(* CODESYS project CÓDIGO FINAL - Separação de caixas coloridas.project

Project tree, tasks and I/O mapping:
  Device : CODESYS Control Win V3, 3S - Smart Software Solutions GmbH, order no. 305021, version 3.5.11.30
    application Application
      libraries: Standard, * (System)
      task MainTask (cyclic, interval t#20ms, priority 1) calls VACUO_01, VACUO_02, PALETIZADOR_01, PALETIZADOR_02, ESTOCAGEM_01, ESTOCAGEM_02
      program VACUO_01 [LD]
      Symbols
      program VACUO_02 [LD]
      global variables MY_GLOBAL
      program PALETIZADOR_01 [LD]
      program PALETIZADOR_02 [LD]
      program ESTOCAGEM_01 [LD]
      program ESTOCAGEM_02 [LD]
*)

// Device/Application/MY_GLOBAL
{attribute 'qualified_only'}
VAR_GLOBAL
// 	VARIAVEL GLOBAL
 	CONTROLE:BOOL;
END_VAR

// Device/Application/VACUO_01
PROGRAM VACUO_01
VAR
// PAINEL DE CONTROLE 
	//ENTRADAS
	_START:BOOL;
	_STOP:BOOL;
	_RESET:BOOL;
	_EMERGENCIA_STOP:BOOL;
	
	//SAIDAS
	START_LIGHT:BOOL;
	STOP_LIGHT:BOOL;
	RESET_LIGHT:BOOL;
	RED: BOOL;
	GREEN: BOOL;
	YELLOW: BOOL;
	CONTAGEM_VERDES:UINT;
	CONTAGEM_DEFEITOS: UINT;
	
// ESTEIRA PRINCIPAL
	//ENTRADAS
	_SENSOR_CAIXA:REAL;
	
	//SAIDAS
	ESTEIRA_PRINCIPAL:BOOL;
	ESTEIRA_PRINCIPAL_1:BOOL;

// ESTEIRA SECUDARIA N 01(VERDE)
	//ENTRADAS
	_SENSOR_SAIDA01:BOOL;
	
	//SAIDAS
	ESTEIRA_SECUDARIA01:BOOL;
	ESTEIRA_CURVA_SECUNDARIA1:BOOL;
	ESTEIRA_CURVA_SECUNDARIA1_1:BOOL;
	ESTEIRA_SAIDA_PALETE1: BOOL;
	
// VACUO N 01
	//ENTRADAS
	_SENSOR_ENTRADA01:BOOL;
	_DETECTED_VACUO01:BOOL;
	
	//SAIDAS
	X1:BOOL;
	Y1:BOOL;
	VACUO_1:BOOL;
	
// AUXILIARES
	CAIXA_VERDE: BOOL;
	A1: BOOL;
	A2: BOOL;
	A3: BOOL;
	A4: BOOL;
	A5: BOOL;
	A6: BOOL;
	A7: BOOL;
	A8: BOOL;
	A9: BOOL;
	A10: BOOL;
	A11: BOOL;

//TEMPORIZADORES
	TON_1A: TON;
	TEMPO_1A: TIME;
	TON_2A: TON;
	TEMPO_2A: TIME;
	TON_3A: TON;
	TEMPO_3A: TIME;
	TON_4A: TON;
	TEMPO_4A: TIME;
	TON_5A: TON;
	TEMPO_5A: TIME;
	TON_6A: TON;
	TEMPO_6A: TIME;
	TON_7A: TON;
	TEMPO_7A: TIME;
	TON_8A: TON;
	TEMPO_8A: TIME;
	TON_9A: TON;
	TEMPO_9A: TIME;
	TON_10A: TON;
	TEMPO_10A: TIME;
	TON_11A: TON;
	TEMPO_11A: TIME;

//CONTADORES
	CTU_1A: CTU;
	CONT_1A: WORD;
	CTU_2A: CTU;
	CONT_2A: WORD;
END_VAR
VAR // added by the converter: edge detectors and wires of the graphical bodies
    _w1, _w2, _w3, _w4, _w5, _w6, _w7, _w8, _w9 : BOOL;
END_VAR

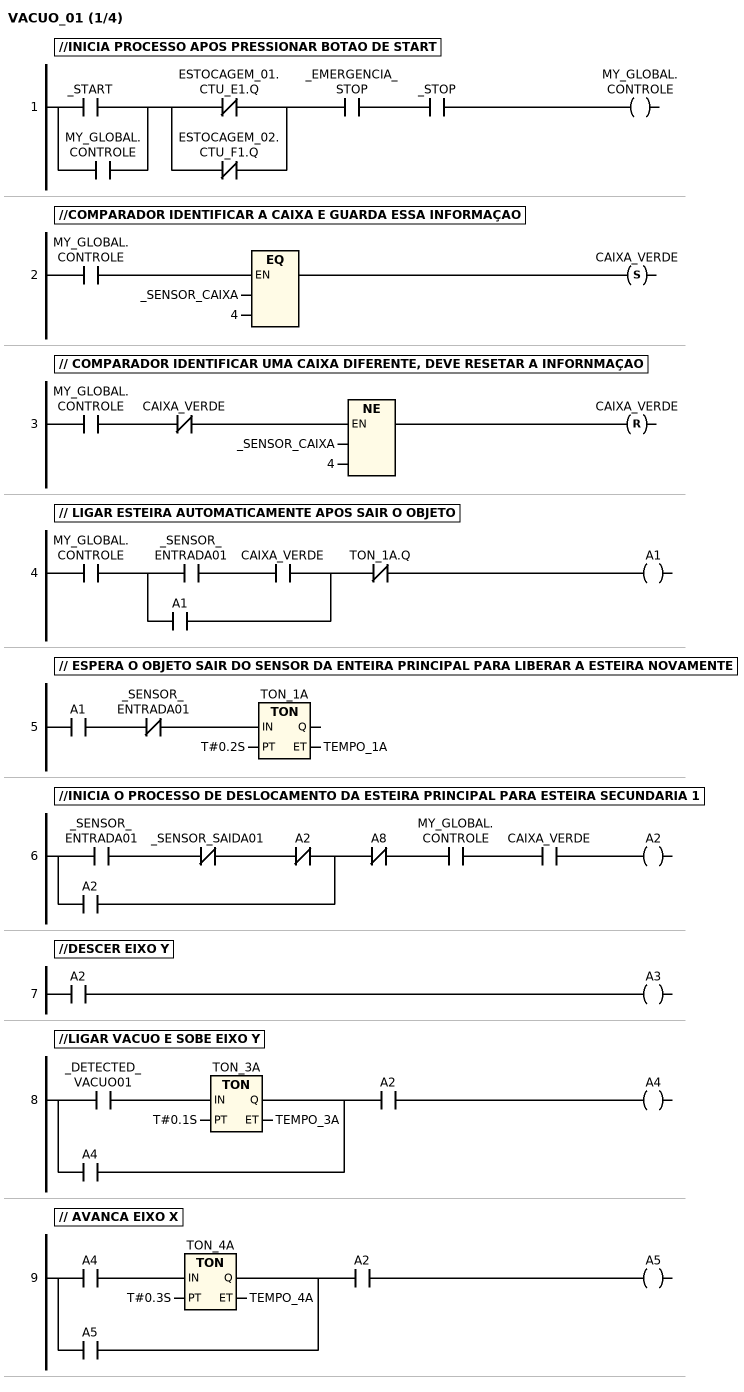
// NETWORK 1
// label: //INICIA PROCESSO APOS PRESSIONAR BOTAO DE START
MY_GLOBAL.CONTROLE := (_START OR MY_GLOBAL.CONTROLE) AND (NOT ESTOCAGEM_01.CTU_E1.Q OR NOT ESTOCAGEM_02.CTU_F1.Q) AND _EMERGENCIA_STOP AND _STOP;

// NETWORK 2
// label: //COMPARADOR IDENTIFICAR A CAIXA E GUARDA ESSA INFORMAÇAO
CAIXA_VERDE S= MY_GLOBAL.CONTROLE AND _SENSOR_CAIXA = 4;

// NETWORK 3
// label: // COMPARADOR IDENTIFICAR UMA CAIXA DIFERENTE, DEVE RESETAR A INFORNMAÇAO
CAIXA_VERDE R= MY_GLOBAL.CONTROLE AND NOT CAIXA_VERDE AND _SENSOR_CAIXA <> 4;

// NETWORK 4
// label: // LIGAR ESTEIRA AUTOMATICAMENTE APOS SAIR O OBJETO
A1 := MY_GLOBAL.CONTROLE AND (_SENSOR_ENTRADA01 AND CAIXA_VERDE OR A1) AND NOT TON_1A.Q;

// NETWORK 5
// label: // ESPERA O OBJETO SAIR DO SENSOR DA ENTEIRA PRINCIPAL PARA LIBERAR A ESTEIRA NOVAMENTE
TON_1A(IN := A1 AND NOT _SENSOR_ENTRADA01, PT := T#0.2S, ET => TEMPO_1A); // TON

// NETWORK 6
// label: //INICIA O PROCESSO DE DESLOCAMENTO DA ESTEIRA PRINCIPAL PARA ESTEIRA SECUNDARIA 1
A2 := (_SENSOR_ENTRADA01 AND NOT _SENSOR_SAIDA01 AND NOT A2 OR A2) AND NOT A8 AND MY_GLOBAL.CONTROLE AND CAIXA_VERDE;

// NETWORK 7
// label: //DESCER EIXO Y
A3 := A2;

// NETWORK 8
// label: //LIGAR VACUO E SOBE EIXO Y
TON_3A(IN := _DETECTED_VACUO01, PT := T#0.1S, ET => TEMPO_3A); // TON
A4 := (TON_3A.Q OR A4) AND A2;

// NETWORK 9
// label: // AVANCA EIXO X
TON_4A(IN := A4, PT := T#0.3S, ET => TEMPO_4A); // TON
A5 := (TON_4A.Q OR A5) AND A2;

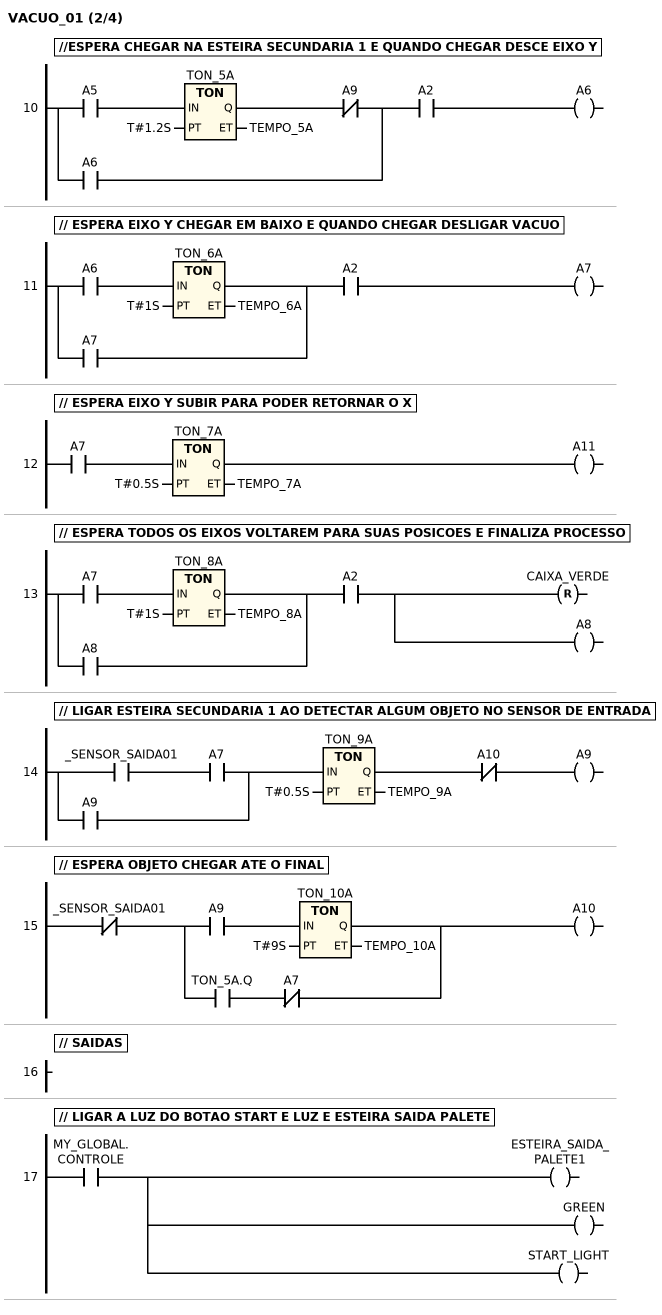
// NETWORK 10
// label: //ESPERA CHEGAR NA ESTEIRA SECUNDARIA 1 E QUANDO CHEGAR DESCE EIXO Y
TON_5A(IN := A5, PT := T#1.2S, ET => TEMPO_5A); // TON
A6 := (TON_5A.Q AND NOT A9 OR A6) AND A2;

// NETWORK 11
// label: // ESPERA EIXO Y CHEGAR EM BAIXO E QUANDO CHEGAR DESLIGAR VACUO
TON_6A(IN := A6, PT := T#1S, ET => TEMPO_6A); // TON
A7 := (TON_6A.Q OR A7) AND A2;

// NETWORK 12
// label: // ESPERA EIXO Y SUBIR PARA PODER RETORNAR O X
TON_7A(IN := A7, PT := T#0.5S, ET => TEMPO_7A); // TON
A11 := TON_7A.Q;

// NETWORK 13
// label: // ESPERA TODOS OS EIXOS VOLTAREM PARA SUAS POSICOES E FINALIZA PROCESSO
TON_8A(IN := A7, PT := T#1S, ET => TEMPO_8A); // TON
_w1 := (TON_8A.Q OR A8) AND A2;
CAIXA_VERDE R= _w1;
A8 := _w1;

// NETWORK 14
// label: // LIGAR ESTEIRA SECUNDARIA 1 AO DETECTAR ALGUM OBJETO NO SENSOR DE ENTRADA
TON_9A(IN := _SENSOR_SAIDA01 AND A7 OR A9, PT := T#0.5S, ET => TEMPO_9A); // TON
A9 := TON_9A.Q AND NOT A10;

// NETWORK 15
// label: // ESPERA OBJETO CHEGAR ATE O FINAL
_w2 := NOT _SENSOR_SAIDA01;
_w3 := (_w2 AND TON_5A.Q) AND NOT A7;
IF NOT _w3 THEN
    TON_10A(IN := _w2 AND A9, PT := T#9S, ET => TEMPO_10A); // TON
    _w3 := TON_10A.Q;
END_IF
A10 := _w3;

// NETWORK 16
// label: // SAIDAS

// NETWORK 17
// label: // LIGAR A LUZ DO BOTAO START E LUZ E ESTEIRA SAIDA PALETE
ESTEIRA_SAIDA_PALETE1 := MY_GLOBAL.CONTROLE;
GREEN := MY_GLOBAL.CONTROLE;
START_LIGHT := MY_GLOBAL.CONTROLE;

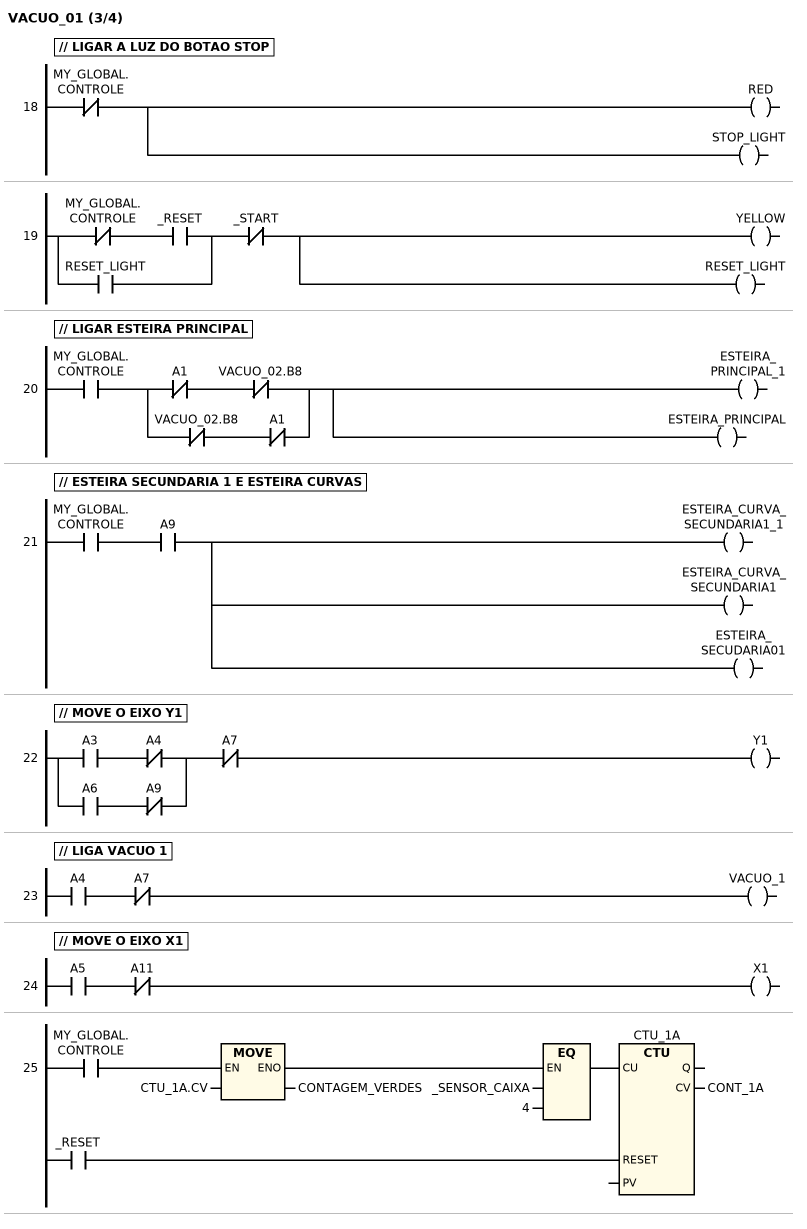
// NETWORK 18
// label: // LIGAR A LUZ DO BOTAO STOP
_w4 := NOT MY_GLOBAL.CONTROLE;
RED := _w4;
STOP_LIGHT := _w4;

// NETWORK 19
_w5 := (NOT MY_GLOBAL.CONTROLE AND _RESET OR RESET_LIGHT) AND NOT _START;
YELLOW := _w5;
RESET_LIGHT := _w5;

// NETWORK 20
// label: // LIGAR ESTEIRA PRINCIPAL
_w6 := MY_GLOBAL.CONTROLE AND (NOT A1 AND NOT VACUO_02.B8 OR NOT VACUO_02.B8 AND NOT A1);
ESTEIRA_PRINCIPAL_1 := _w6;
ESTEIRA_PRINCIPAL := _w6;

// NETWORK 21
// label: // ESTEIRA SECUNDARIA 1 E ESTEIRA CURVAS
_w7 := MY_GLOBAL.CONTROLE AND A9;
ESTEIRA_CURVA_SECUNDARIA1_1 := _w7;
ESTEIRA_CURVA_SECUNDARIA1 := _w7;
ESTEIRA_SECUDARIA01 := _w7;

// NETWORK 22
// label: // MOVE O EIXO Y1
Y1 := (A3 AND NOT A4 OR A6 AND NOT A9) AND NOT A7;

// NETWORK 23
// label: // LIGA VACUO 1
VACUO_1 := A4 AND NOT A7;

// NETWORK 24
// label: // MOVE O EIXO X1
X1 := A5 AND NOT A11;

// NETWORK 25
_w8 := MY_GLOBAL.CONTROLE;
IF _w8 THEN CONTAGEM_VERDES := CTU_1A.CV; END_IF
CTU_1A(CU := _w8 AND _SENSOR_CAIXA = 4, RESET := _RESET, CV => CONT_1A); // CTU

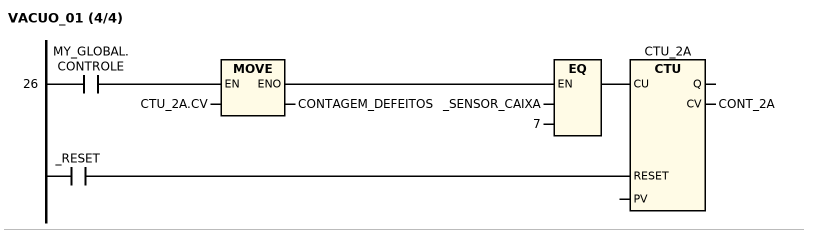
// NETWORK 26
_w9 := MY_GLOBAL.CONTROLE;
IF _w9 THEN CONTAGEM_DEFEITOS := CTU_2A.CV; END_IF
CTU_2A(CU := _w9 AND _SENSOR_CAIXA = 7, RESET := _RESET, CV => CONT_2A); // CTU

END_PROGRAM

// Device/Application/ESTOCAGEM_01
PROGRAM ESTOCAGEM_01
VAR
//ENTRADA
	_SENSOR_ESTOCAGEM1: BOOL;

//SAIDA
	CRANE_ENTRADA1:BOOL;
	CRANE_SAIDA1:BOOL;
	CRANE_SUBIR1:BOOL;
	ESTEIRA_ESTOCAGEM1:BOOL;
	ESTEIRA_MEIO_ESTOCAGEM1:BOOL;
	ESTEIRA_CURVA_ESTOCAGEM1:BOOL;
	POSICAO: UINT;
//AUXILIARES	
	E1: BOOL;
	E2: BOOL;
	E3: BOOL;
	E4: BOOL;
	E5: BOOL;	

//TEMPORIZAODES 
	TON_E1: TON;
	TEMPO_E1: TIME;
	TON_E2: TON;
	TEMPO_E2: TIME;
	TON_E3: TON;
	TEMPO_E3: TIME;
	TON_E4: TON;
	TEMPO_E4: TIME;
	TON_E5: TON;
	TEMPO_E5: TIME;
	TON_E6: TON;
	TEMPO_E6: TIME;

//CONTADORES
	CTU_E1: CTU;
	CONT_E1: WORD;

// TEMPORIZADORES DE CADA PRATILEIRA
	TON_1:TON;
	TEMPO_1:TIME;
	TON_2:TON;
	TEMPO_2:TIME;
	TON_3:TON;
	TEMPO_3: TIME;
	TON_4:TON;
	TEMPO_4:TIME;
	TON_5:TON;
	TEMPO_5:TIME;
	TON_6:TON;
	TEMPO_6:TIME;
	TON_7:TON;
	TEMPO_7:TIME;
	TON_8:TON;
	TEMPO_8:TIME;
	TON_9:TON;
	TEMPO_9:TIME;
	TON_10: TON;
	TEMPO_10: TIME;
	TON_11: TON;
	TEMPO_11: TIME;
	TON_12: TON;
	TEMPO_12: TIME;
	TON_13:TON;
	TEMPO_13: TIME;
	TON_14: TON;
	TEMPO_14: TIME;
	TON_15: TON;
	TEMPO_15: TIME;
	TON_16: TON;
	TEMPO_16: TIME;
	TON_17: TON;
	TEMPO_17: TIME;
	TON_18: TON;
	TEMPO_18: TIME;
	TON_19: TON;
	TEMPO_19: TIME;
	TON_20: TON;
	TEMPO_20: TIME;
	TON_21: TON;
	TEMPO_21: TIME;
	TON_22: TON;
	TEMPO_22: TIME;
	TON_23: TON;
	TEMPO_23: TIME;
	TON_24: TON;
	TEMPO_24: TIME;
	TON_25: TON;
	TEMPO_25: TIME;
	TON_26: TON;
	TEMPO_26: TIME;
	TON_27: TON;
	TEMPO_27: TIME;
	TON_28: TON;
	TEMPO_28: TIME;
	TON_29: TON;
	TEMPO_29: TIME;
	TON_30: TON;
	TEMPO_30: TIME;
	TON_31: TON;
	TEMPO_31: TIME;
	TON_32: TON;
	TEMPO_32: TIME;
	TON_33: TON;
	TEMPO_33: TIME;
	TON_34: TON;
	TEMPO_34: TIME;
	TON_35: TON;
	TEMPO_35: TIME;
	TON_36: TON;
	TEMPO_36: TIME;
	TON_37: TON;
	TEMPO_37: TIME;
	TON_38: TON;
	TEMPO_38: TIME;
	TON_39: TON;
	TEMPO_39: TIME;
	TON_40: TON;
	TEMPO_40: TIME;
	TON_41: TON;
	TEMPO_41: TIME;
	TON_42: TON;
	TEMPO_42: TIME;
	TON_43: TON;
	TEMPO_43: TIME;
	TON_44: TON;
	TEMPO_44: TIME;
	TON_45: TON;
	TEMPO_45: TIME;
	TON_46: TON;
	TEMPO_46: TIME;
	TON_47: TON;
	TEMPO_47: TIME;
	TON_48: TON;
	TEMPO_48: TIME;
	TON_49: TON;
	TEMPO_49: TIME;
	TON_50: TON;
	TEMPO_50: TIME;
	TON_51: TON;
	TEMPO_51: TIME;
	TON_52: TON;
	TEMPO_52: TIME;
	TON_53: TON;
	TEMPO_53: TIME;
	TON_54: TON;
	TEMPO_54: TIME;

// AUXILIARES DE CADA PRATILEIRA
	T1:BOOL;
	T2:BOOL;
	T3:BOOL;
	T4:BOOL;
	T5:BOOL;
	T6:BOOL;
	T7:BOOL;
	T8:BOOL;
	T9:BOOL;
	T10:BOOL;
	T11:BOOL;
	T12:BOOL;
	T13:BOOL;
	T14:BOOL;
	T15:BOOL;
	T16:BOOL;
	T17:BOOL;
	T18:BOOL;	
	T19:BOOL;
	T20:BOOL;
	T21:BOOL;
	T22:BOOL;
	T23: BOOL;
	T24: BOOL;
	T25: BOOL;
	T26: BOOL;
	T27: BOOL;
	T28: BOOL;
	T29: BOOL;
	T30: BOOL;
	T31: BOOL;
	T32: BOOL;
	T33: BOOL;
	T34: BOOL;
	T35: BOOL;
	T36: BOOL;
	T37: BOOL;
	T38: BOOL;
	T39: BOOL;
	T40: BOOL;
	T41: BOOL;
	T42: BOOL;
	T43: BOOL;
	T44: BOOL;
	T45: BOOL;
	T46: BOOL;
	T47: BOOL;
	T48: BOOL;
	T49: BOOL;
	T50: BOOL;
	T51: BOOL;
	T52: BOOL;
	T53: BOOL;
	T54: BOOL;
	T55: BOOL;
END_VAR
VAR // added by the converter: edge detectors and wires of the graphical bodies
    _w1, _w2, _w3 : BOOL;
END_VAR

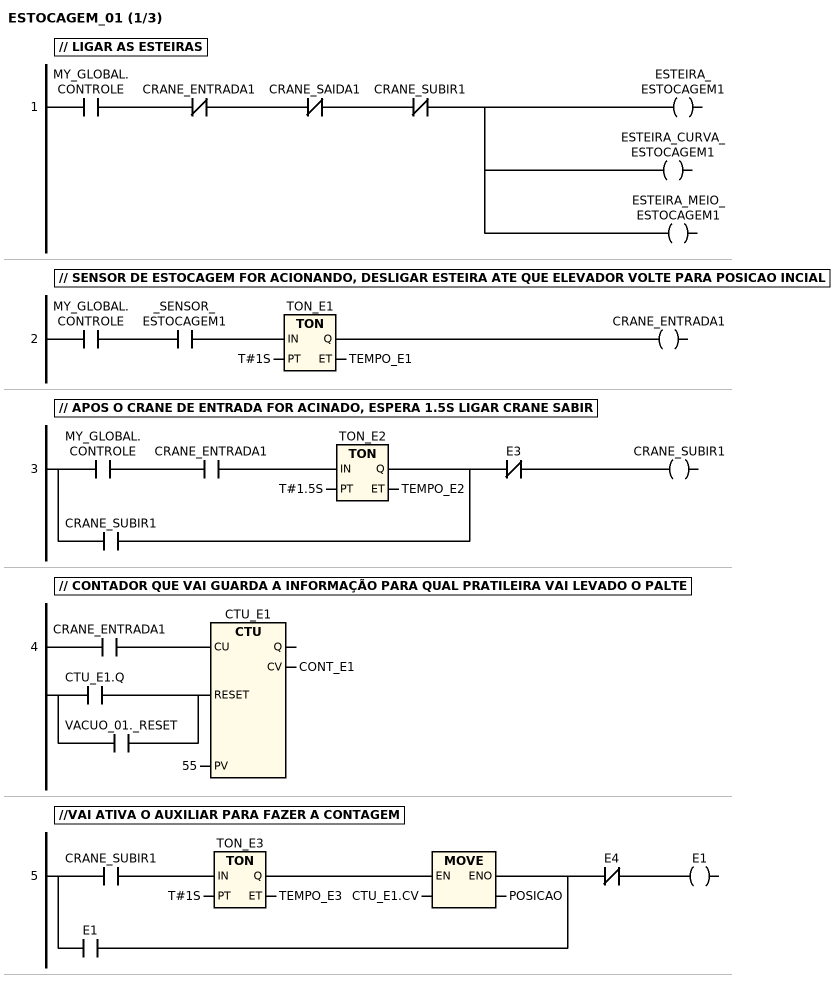
// NETWORK 1
// label: // LIGAR AS ESTEIRAS
_w1 := MY_GLOBAL.CONTROLE AND NOT CRANE_ENTRADA1 AND NOT CRANE_SAIDA1 AND NOT CRANE_SUBIR1;
ESTEIRA_ESTOCAGEM1 := _w1;
ESTEIRA_CURVA_ESTOCAGEM1 := _w1;
ESTEIRA_MEIO_ESTOCAGEM1 := _w1;

// NETWORK 2
// label: // SENSOR DE ESTOCAGEM FOR ACIONANDO, DESLIGAR ESTEIRA ATE QUE ELEVADOR VOLTE PARA POSICAO INCIAL
TON_E1(IN := MY_GLOBAL.CONTROLE AND _SENSOR_ESTOCAGEM1, PT := T#1S, ET => TEMPO_E1); // TON
CRANE_ENTRADA1 := TON_E1.Q;

// NETWORK 3
// label: // APOS O CRANE DE ENTRADA FOR ACINADO, ESPERA 1.5S LIGAR CRANE SABIR
TON_E2(IN := MY_GLOBAL.CONTROLE AND CRANE_ENTRADA1, PT := T#1.5S, ET => TEMPO_E2); // TON
CRANE_SUBIR1 := (TON_E2.Q OR CRANE_SUBIR1) AND NOT E3;

// NETWORK 4
// label: // CONTADOR QUE VAI GUARDA A INFORMAÇÃO PARA QUAL PRATILEIRA VAI LEVADO O PALTE
CTU_E1(CU := CRANE_ENTRADA1, RESET := CTU_E1.Q OR VACUO_01._RESET, PV := 55, CV => CONT_E1); // CTU

// NETWORK 5
// label: //VAI ATIVA O AUXILIAR PARA FAZER A CONTAGEM
TON_E3(IN := CRANE_SUBIR1, PT := T#1S, ET => TEMPO_E3); // TON
_w2 := TON_E3.Q;
IF _w2 THEN POSICAO := CTU_E1.CV; END_IF
E1 := (_w2 OR E1) AND NOT E4;

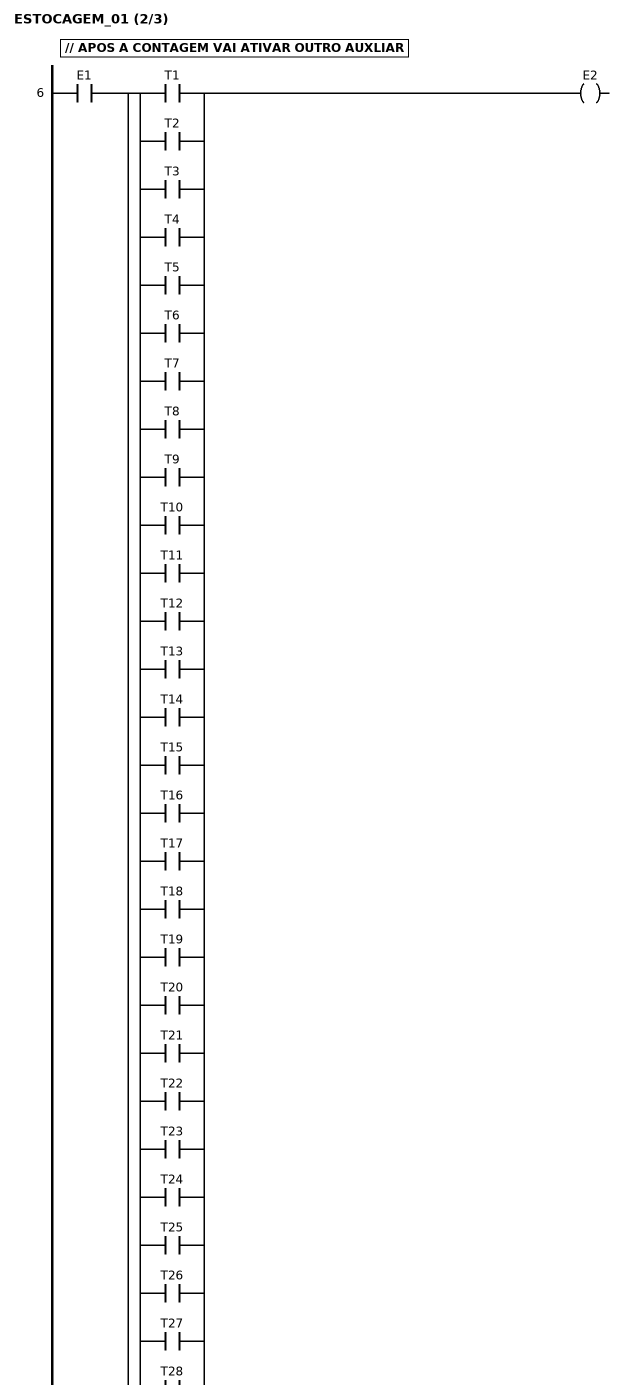
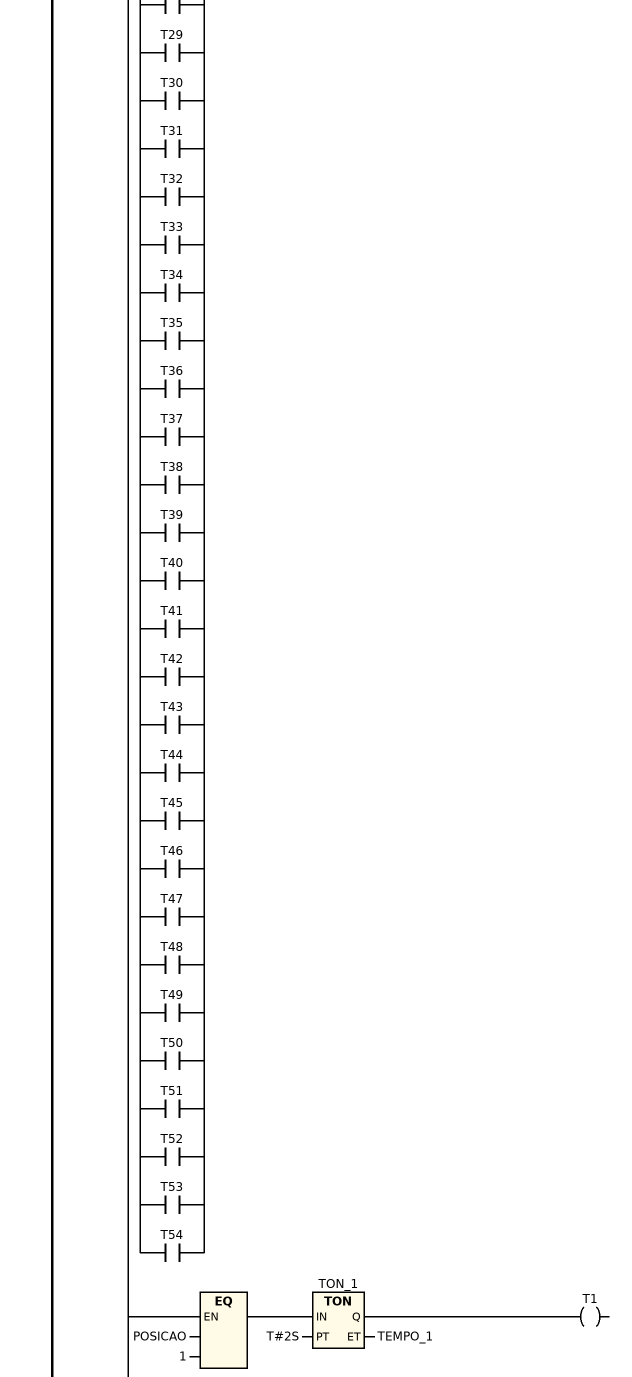
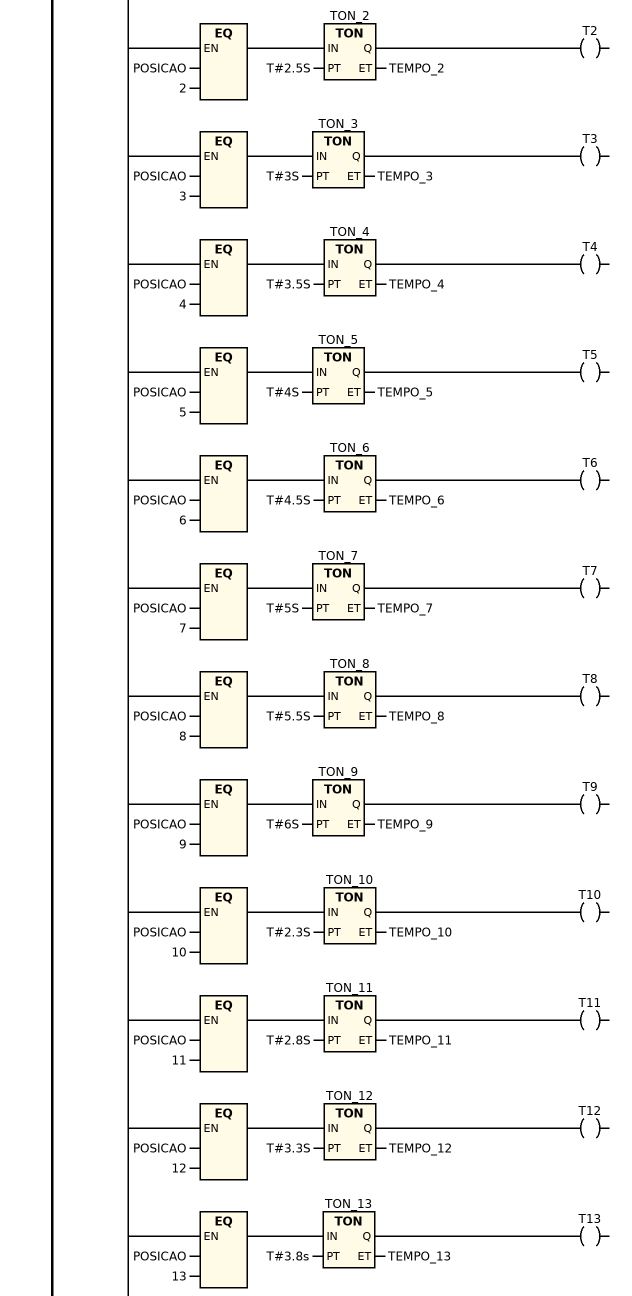
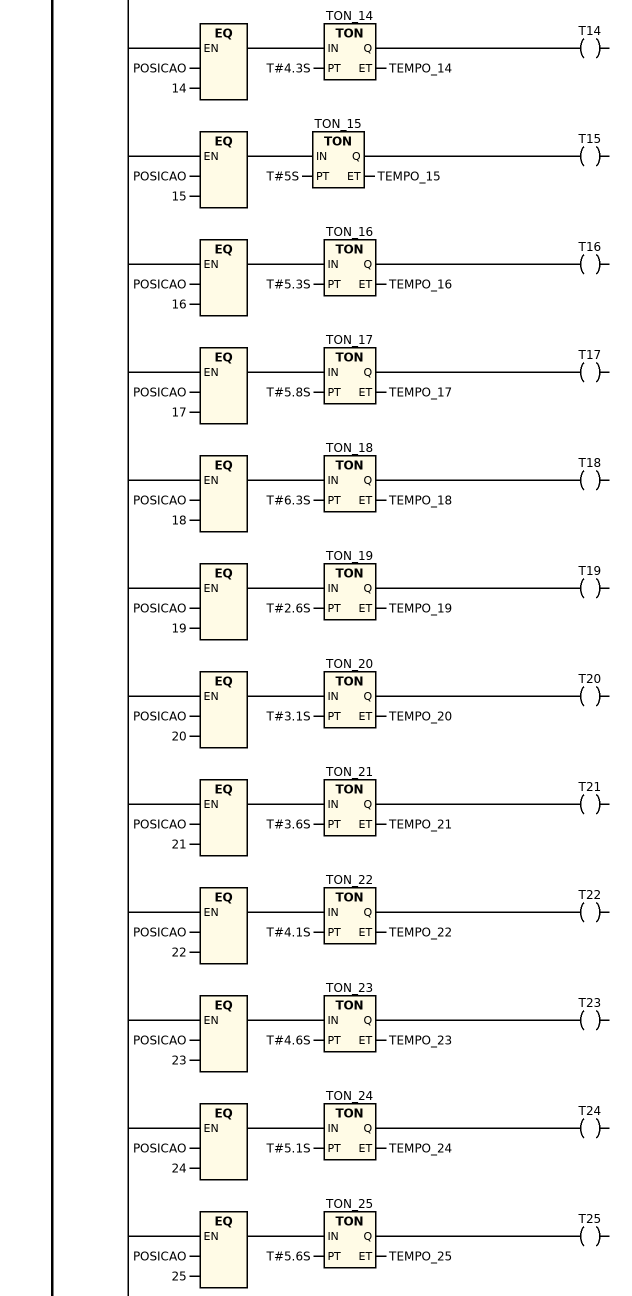
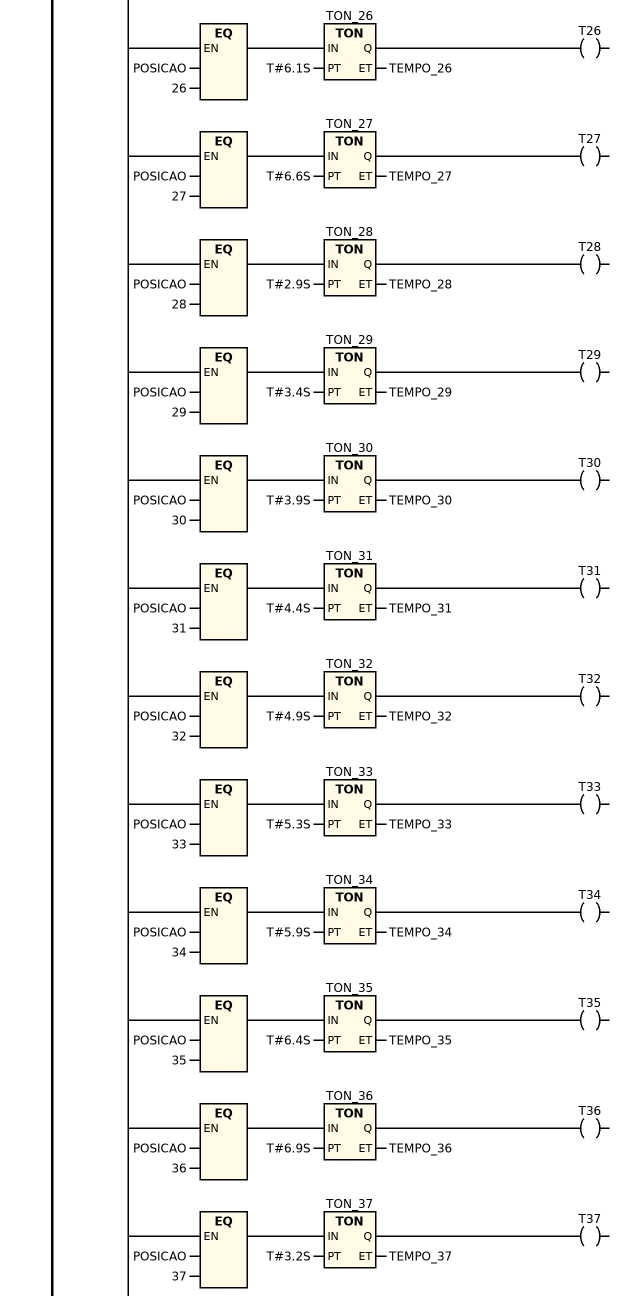
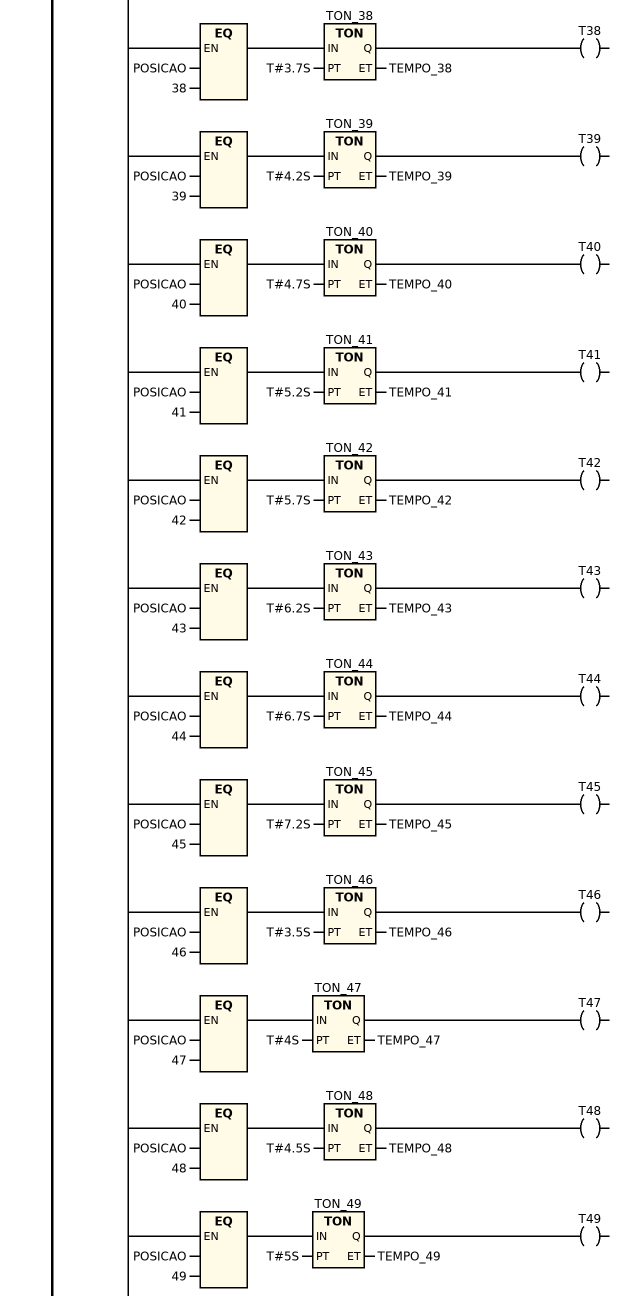
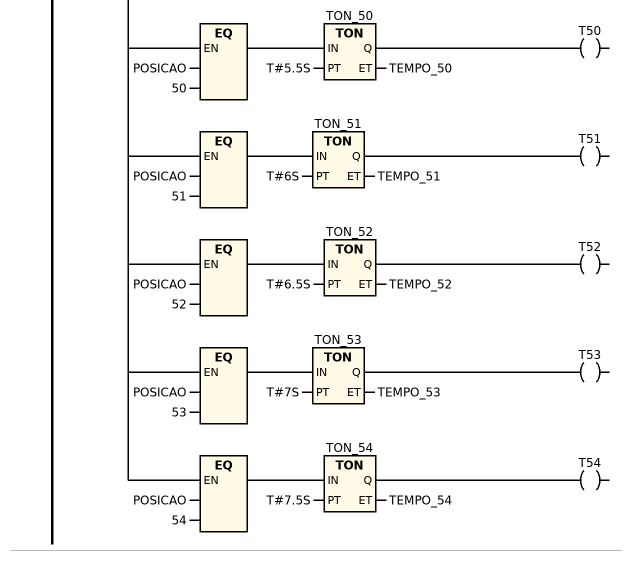
// NETWORK 6
// label: // APOS A CONTAGEM VAI ATIVAR OUTRO AUXLIAR
E2 := E1 AND (T1 OR T2 OR T3 OR T4 OR T5 OR T6 OR T7 OR T8 OR T9 OR T10 OR T11 OR T12 OR T13 OR T14 OR T15 OR T16 OR T17 OR T18 OR T19 OR T20 OR T21 OR T22 OR T23 OR T24 OR T25 OR T26 OR T27 OR T28 OR T29 OR T30 OR T31 OR T32 OR T33 OR T34 OR T35 OR T36 OR T37 OR T38 OR T39 OR T40 OR T41 OR T42 OR T43 OR T44 OR T45 OR T46 OR T47 OR T48 OR T49 OR T50 OR T51 OR T52 OR T53 OR T54);
TON_1(IN := E1 AND POSICAO = 1, PT := T#2S, ET => TEMPO_1); // TON
T1 := TON_1.Q;
TON_2(IN := E1 AND POSICAO = 2, PT := T#2.5S, ET => TEMPO_2); // TON
T2 := TON_2.Q;
TON_3(IN := E1 AND POSICAO = 3, PT := T#3S, ET => TEMPO_3); // TON
T3 := TON_3.Q;
TON_4(IN := E1 AND POSICAO = 4, PT := T#3.5S, ET => TEMPO_4); // TON
T4 := TON_4.Q;
TON_5(IN := E1 AND POSICAO = 5, PT := T#4S, ET => TEMPO_5); // TON
T5 := TON_5.Q;
TON_6(IN := E1 AND POSICAO = 6, PT := T#4.5S, ET => TEMPO_6); // TON
T6 := TON_6.Q;
TON_7(IN := E1 AND POSICAO = 7, PT := T#5S, ET => TEMPO_7); // TON
T7 := TON_7.Q;
TON_8(IN := E1 AND POSICAO = 8, PT := T#5.5S, ET => TEMPO_8); // TON
T8 := TON_8.Q;
TON_9(IN := E1 AND POSICAO = 9, PT := T#6S, ET => TEMPO_9); // TON
T9 := TON_9.Q;
TON_10(IN := E1 AND POSICAO = 10, PT := T#2.3S, ET => TEMPO_10); // TON
T10 := TON_10.Q;
TON_11(IN := E1 AND POSICAO = 11, PT := T#2.8S, ET => TEMPO_11); // TON
T11 := TON_11.Q;
TON_12(IN := E1 AND POSICAO = 12, PT := T#3.3S, ET => TEMPO_12); // TON
T12 := TON_12.Q;
TON_13(IN := E1 AND POSICAO = 13, PT := T#3.8s, ET => TEMPO_13); // TON
T13 := TON_13.Q;
TON_14(IN := E1 AND POSICAO = 14, PT := T#4.3S, ET => TEMPO_14); // TON
T14 := TON_14.Q;
TON_15(IN := E1 AND POSICAO = 15, PT := T#5S, ET => TEMPO_15); // TON
T15 := TON_15.Q;
TON_16(IN := E1 AND POSICAO = 16, PT := T#5.3S, ET => TEMPO_16); // TON
T16 := TON_16.Q;
TON_17(IN := E1 AND POSICAO = 17, PT := T#5.8S, ET => TEMPO_17); // TON
T17 := TON_17.Q;
TON_18(IN := E1 AND POSICAO = 18, PT := T#6.3S, ET => TEMPO_18); // TON
T18 := TON_18.Q;
TON_19(IN := E1 AND POSICAO = 19, PT := T#2.6S, ET => TEMPO_19); // TON
T19 := TON_19.Q;
TON_20(IN := E1 AND POSICAO = 20, PT := T#3.1S, ET => TEMPO_20); // TON
T20 := TON_20.Q;
TON_21(IN := E1 AND POSICAO = 21, PT := T#3.6S, ET => TEMPO_21); // TON
T21 := TON_21.Q;
TON_22(IN := E1 AND POSICAO = 22, PT := T#4.1S, ET => TEMPO_22); // TON
T22 := TON_22.Q;
TON_23(IN := E1 AND POSICAO = 23, PT := T#4.6S, ET => TEMPO_23); // TON
T23 := TON_23.Q;
TON_24(IN := E1 AND POSICAO = 24, PT := T#5.1S, ET => TEMPO_24); // TON
T24 := TON_24.Q;
TON_25(IN := E1 AND POSICAO = 25, PT := T#5.6S, ET => TEMPO_25); // TON
T25 := TON_25.Q;
TON_26(IN := E1 AND POSICAO = 26, PT := T#6.1S, ET => TEMPO_26); // TON
T26 := TON_26.Q;
TON_27(IN := E1 AND POSICAO = 27, PT := T#6.6S, ET => TEMPO_27); // TON
T27 := TON_27.Q;
TON_28(IN := E1 AND POSICAO = 28, PT := T#2.9S, ET => TEMPO_28); // TON
T28 := TON_28.Q;
TON_29(IN := E1 AND POSICAO = 29, PT := T#3.4S, ET => TEMPO_29); // TON
T29 := TON_29.Q;
TON_30(IN := E1 AND POSICAO = 30, PT := T#3.9S, ET => TEMPO_30); // TON
T30 := TON_30.Q;
TON_31(IN := E1 AND POSICAO = 31, PT := T#4.4S, ET => TEMPO_31); // TON
T31 := TON_31.Q;
TON_32(IN := E1 AND POSICAO = 32, PT := T#4.9S, ET => TEMPO_32); // TON
T32 := TON_32.Q;
TON_33(IN := E1 AND POSICAO = 33, PT := T#5.3S, ET => TEMPO_33); // TON
T33 := TON_33.Q;
TON_34(IN := E1 AND POSICAO = 34, PT := T#5.9S, ET => TEMPO_34); // TON
T34 := TON_34.Q;
TON_35(IN := E1 AND POSICAO = 35, PT := T#6.4S, ET => TEMPO_35); // TON
T35 := TON_35.Q;
TON_36(IN := E1 AND POSICAO = 36, PT := T#6.9S, ET => TEMPO_36); // TON
T36 := TON_36.Q;
TON_37(IN := E1 AND POSICAO = 37, PT := T#3.2S, ET => TEMPO_37); // TON
T37 := TON_37.Q;
TON_38(IN := E1 AND POSICAO = 38, PT := T#3.7S, ET => TEMPO_38); // TON
T38 := TON_38.Q;
TON_39(IN := E1 AND POSICAO = 39, PT := T#4.2S, ET => TEMPO_39); // TON
T39 := TON_39.Q;
TON_40(IN := E1 AND POSICAO = 40, PT := T#4.7S, ET => TEMPO_40); // TON
T40 := TON_40.Q;
TON_41(IN := E1 AND POSICAO = 41, PT := T#5.2S, ET => TEMPO_41); // TON
T41 := TON_41.Q;
TON_42(IN := E1 AND POSICAO = 42, PT := T#5.7S, ET => TEMPO_42); // TON
T42 := TON_42.Q;
TON_43(IN := E1 AND POSICAO = 43, PT := T#6.2S, ET => TEMPO_43); // TON
T43 := TON_43.Q;
TON_44(IN := E1 AND POSICAO = 44, PT := T#6.7S, ET => TEMPO_44); // TON
T44 := TON_44.Q;
TON_45(IN := E1 AND POSICAO = 45, PT := T#7.2S, ET => TEMPO_45); // TON
T45 := TON_45.Q;
TON_46(IN := E1 AND POSICAO = 46, PT := T#3.5S, ET => TEMPO_46); // TON
T46 := TON_46.Q;
TON_47(IN := E1 AND POSICAO = 47, PT := T#4S, ET => TEMPO_47); // TON
T47 := TON_47.Q;
TON_48(IN := E1 AND POSICAO = 48, PT := T#4.5S, ET => TEMPO_48); // TON
T48 := TON_48.Q;
TON_49(IN := E1 AND POSICAO = 49, PT := T#5S, ET => TEMPO_49); // TON
T49 := TON_49.Q;
TON_50(IN := E1 AND POSICAO = 50, PT := T#5.5S, ET => TEMPO_50); // TON
T50 := TON_50.Q;
TON_51(IN := E1 AND POSICAO = 51, PT := T#6S, ET => TEMPO_51); // TON
T51 := TON_51.Q;
TON_52(IN := E1 AND POSICAO = 52, PT := T#6.5S, ET => TEMPO_52); // TON
T52 := TON_52.Q;
TON_53(IN := E1 AND POSICAO = 53, PT := T#7S, ET => TEMPO_53); // TON
T53 := TON_53.Q;
TON_54(IN := E1 AND POSICAO = 54, PT := T#7.5S, ET => TEMPO_54); // TON
T54 := TON_54.Q;

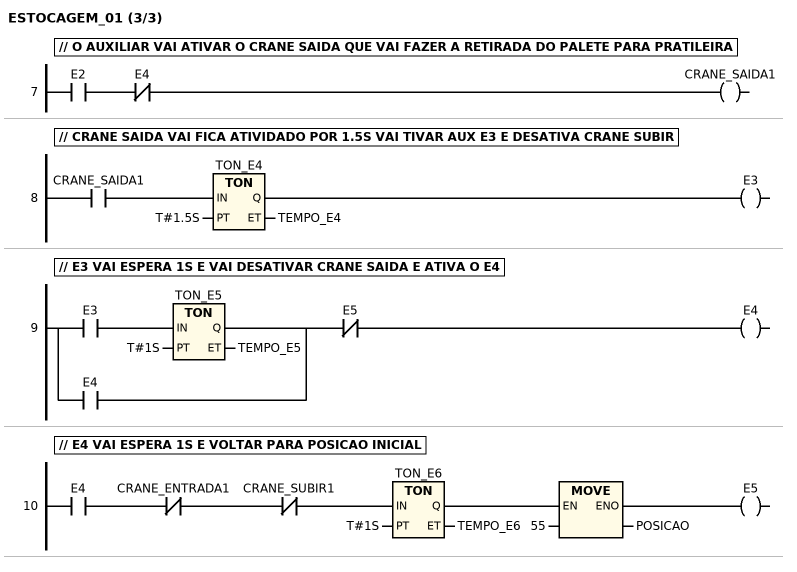
// NETWORK 7
// label: // O AUXILIAR VAI ATIVAR O CRANE SAIDA QUE VAI FAZER A RETIRADA DO PALETE PARA PRATILEIRA
CRANE_SAIDA1 := E2 AND NOT E4;

// NETWORK 8
// label: // CRANE SAIDA VAI FICA ATIVIDADO POR 1.5S VAI TIVAR AUX E3 E DESATIVA CRANE SUBIR
TON_E4(IN := CRANE_SAIDA1, PT := T#1.5S, ET => TEMPO_E4); // TON
E3 := TON_E4.Q;

// NETWORK 9
// label: // E3 VAI ESPERA 1S E VAI DESATIVAR CRANE SAIDA E ATIVA O E4
TON_E5(IN := E3, PT := T#1S, ET => TEMPO_E5); // TON
E4 := (TON_E5.Q OR E4) AND NOT E5;

// NETWORK 10
// label: // E4 VAI ESPERA 1S E VOLTAR PARA POSICAO INICIAL
TON_E6(IN := E4 AND NOT CRANE_ENTRADA1 AND NOT CRANE_SUBIR1, PT := T#1S, ET => TEMPO_E6); // TON
_w3 := TON_E6.Q;
IF _w3 THEN POSICAO := 55; END_IF
E5 := _w3;

END_PROGRAM

// Device/Application/ESTOCAGEM_02
PROGRAM ESTOCAGEM_02
VAR
//ENTRADA
	_SENSOR_ESTOCAGEM2: BOOL;

//SAIDA
	CRANE_ENTRADA2:BOOL;
	CRANE_SAIDA2:BOOL;
	CRANE_SUBIR2:BOOL;
	ESTEIRA_ESTOCAGEM2:BOOL;
	ESTEIRA_MEIO_ESTOCAGEM2:BOOL;
	ESTEIRA_MEIO_ESTOCAGEM2_1:BOOL;
	ESTEIRA_CURVA_ESTOCAGEM2:BOOL;
	POSICAO: UINT;
	
//AUXILIARES	
	F1: BOOL;
	F2: BOOL;
	F3: BOOL;
	F4: BOOL;
	F5: BOOL;	

//TEMPORIZAODES 
	TON_F1: TON;
	TEMPO_F1: TIME;
	TON_F2: TON;
	TEMPO_F2: TIME;
	TON_F3: TON;
	TEMPO_F3: TIME;
	TON_F4: TON;
	TEMPO_F4: TIME;
	TON_F5: TON;
	TEMPO_F5: TIME;
	TON_F6: TON;
	TEMPO_F6: TIME;

//CONTADORES
	CTU_F1: CTU;
	CONT_F1: WORD;

// TEMPORIZADORES DE CADA LUGAR
	TON_1:TON;
	TEMPO_1:TIME;
	TON_2:TON;
	TEMPO_2:TIME;
	TON_3:TON;
	TEMPO_3: TIME;
	TON_4:TON;
	TEMPO_4:TIME;
	TON_5:TON;
	TEMPO_5:TIME;
	TON_6:TON;
	TEMPO_6:TIME;
	TON_7:TON;
	TEMPO_7:TIME;
	TON_8:TON;
	TEMPO_8:TIME;
	TON_9:TON;
	TEMPO_9:TIME;
	TON_10: TON;
	TEMPO_10: TIME;
	TON_11: TON;
	TEMPO_11: TIME;
	TON_12: TON;
	TEMPO_12: TIME;
	TON_13:TON;
	TEMPO_13: TIME;
	TON_14: TON;
	TEMPO_14: TIME;
	TON_15: TON;
	TEMPO_15: TIME;
	TON_16: TON;
	TEMPO_16: TIME;
	TON_17: TON;
	TEMPO_17: TIME;
	TON_18: TON;
	TEMPO_18: TIME;
	TON_19: TON;
	TEMPO_19: TIME;
	TON_20: TON;
	TEMPO_20: TIME;
	TON_21: TON;
	TEMPO_21: TIME;
	TON_22: TON;
	TEMPO_22: TIME;
	TON_23: TON;
	TEMPO_23: TIME;
	TON_24: TON;
	TEMPO_24: TIME;
	TON_25: TON;
	TEMPO_25: TIME;
	TON_26: TON;
	TEMPO_26: TIME;
	TON_27: TON;
	TEMPO_27: TIME;
	TON_28: TON;
	TEMPO_28: TIME;
	TON_29: TON;
	TEMPO_29: TIME;
	TON_30: TON;
	TEMPO_30: TIME;
	TON_31: TON;
	TEMPO_31: TIME;
	TON_32: TON;
	TEMPO_32: TIME;
	TON_33: TON;
	TEMPO_33: TIME;
	TON_34: TON;
	TEMPO_34: TIME;
	TON_35: TON;
	TEMPO_35: TIME;
	TON_36: TON;
	TEMPO_36: TIME;
	TON_37: TON;
	TEMPO_37: TIME;
	TON_38: TON;
	TEMPO_38: TIME;
	TON_39: TON;
	TEMPO_39: TIME;
	TON_40: TON;
	TEMPO_40: TIME;
	TON_41: TON;
	TEMPO_41: TIME;
	TON_42: TON;
	TEMPO_42: TIME;
	TON_43: TON;
	TEMPO_43: TIME;
	TON_44: TON;
	TEMPO_44: TIME;
	TON_45: TON;
	TEMPO_45: TIME;
	TON_46: TON;
	TEMPO_46: TIME;
	TON_47: TON;
	TEMPO_47: TIME;
	TON_48: TON;
	TEMPO_48: TIME;
	TON_49: TON;
	TEMPO_49: TIME;
	TON_50: TON;
	TEMPO_50: TIME;
	TON_51: TON;
	TEMPO_51: TIME;
	TON_52: TON;
	TEMPO_52: TIME;
	TON_53: TON;
	TEMPO_53: TIME;
	TON_54: TON;
	TEMPO_54: TIME;

// AUXILIARES DE CADA LUGAR
	T1:BOOL;
	T2:BOOL;
	T3:BOOL;
	T4:BOOL;
	T5:BOOL;
	T6:BOOL;
	T7:BOOL;
	T8:BOOL;
	T9:BOOL;
	T10:BOOL;
	T11:BOOL;
	T12:BOOL;
	T13:BOOL;
	T14:BOOL;
	T15:BOOL;
	T16:BOOL;
	T17:BOOL;
	T18:BOOL;	
	T19:BOOL;
	T20:BOOL;
	T21:BOOL;
	T22:BOOL;
	T23: BOOL;
	T24: BOOL;
	T25: BOOL;
	T26: BOOL;
	T27: BOOL;
	T28: BOOL;
	T29: BOOL;
	T30: BOOL;
	T31: BOOL;
	T32: BOOL;
	T33: BOOL;
	T34: BOOL;
	T35: BOOL;
	T36: BOOL;
	T37: BOOL;
	T38: BOOL;
	T39: BOOL;
	T40: BOOL;
	T41: BOOL;
	T42: BOOL;
	T43: BOOL;
	T44: BOOL;
	T45: BOOL;
	T46: BOOL;
	T47: BOOL;
	T48: BOOL;
	T49: BOOL;
	T50: BOOL;
	T51: BOOL;
	T52: BOOL;
	T53: BOOL;
	T54: BOOL;
	T55: BOOL;
END_VAR
VAR // added by the converter: edge detectors and wires of the graphical bodies
    _w1, _w2, _w3 : BOOL;
END_VAR

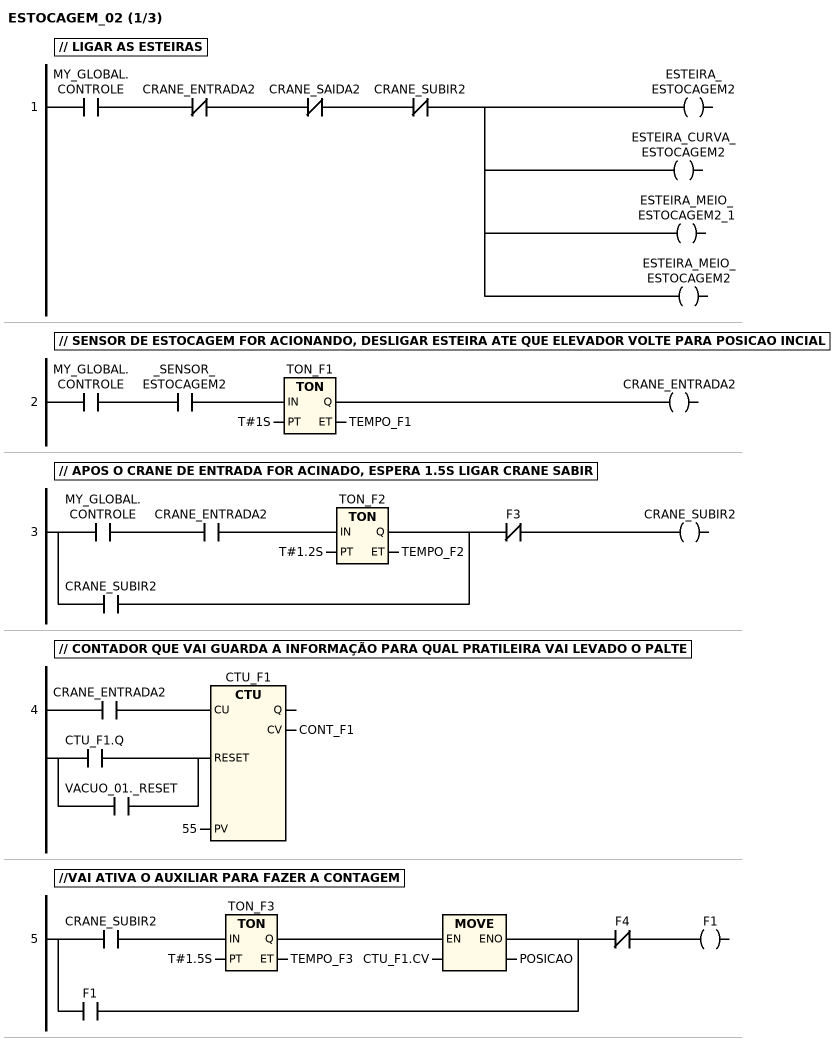
// NETWORK 1
// label: // LIGAR AS ESTEIRAS
_w1 := MY_GLOBAL.CONTROLE AND NOT CRANE_ENTRADA2 AND NOT CRANE_SAIDA2 AND NOT CRANE_SUBIR2;
ESTEIRA_ESTOCAGEM2 := _w1;
ESTEIRA_CURVA_ESTOCAGEM2 := _w1;
ESTEIRA_MEIO_ESTOCAGEM2_1 := _w1;
ESTEIRA_MEIO_ESTOCAGEM2 := _w1;

// NETWORK 2
// label: // SENSOR DE ESTOCAGEM FOR ACIONANDO, DESLIGAR ESTEIRA ATE QUE ELEVADOR VOLTE PARA POSICAO INCIAL
TON_F1(IN := MY_GLOBAL.CONTROLE AND _SENSOR_ESTOCAGEM2, PT := T#1S, ET => TEMPO_F1); // TON
CRANE_ENTRADA2 := TON_F1.Q;

// NETWORK 3
// label: // APOS O CRANE DE ENTRADA FOR ACINADO, ESPERA 1.5S LIGAR CRANE SABIR
TON_F2(IN := MY_GLOBAL.CONTROLE AND CRANE_ENTRADA2, PT := T#1.2S, ET => TEMPO_F2); // TON
CRANE_SUBIR2 := (TON_F2.Q OR CRANE_SUBIR2) AND NOT F3;

// NETWORK 4
// label: // CONTADOR QUE VAI GUARDA A INFORMAÇÃO PARA QUAL PRATILEIRA VAI LEVADO O PALTE
CTU_F1(CU := CRANE_ENTRADA2, RESET := CTU_F1.Q OR VACUO_01._RESET, PV := 55, CV => CONT_F1); // CTU

// NETWORK 5
// label: //VAI ATIVA O AUXILIAR PARA FAZER A CONTAGEM
TON_F3(IN := CRANE_SUBIR2, PT := T#1.5S, ET => TEMPO_F3); // TON
_w2 := TON_F3.Q;
IF _w2 THEN POSICAO := CTU_F1.CV; END_IF
F1 := (_w2 OR F1) AND NOT F4;

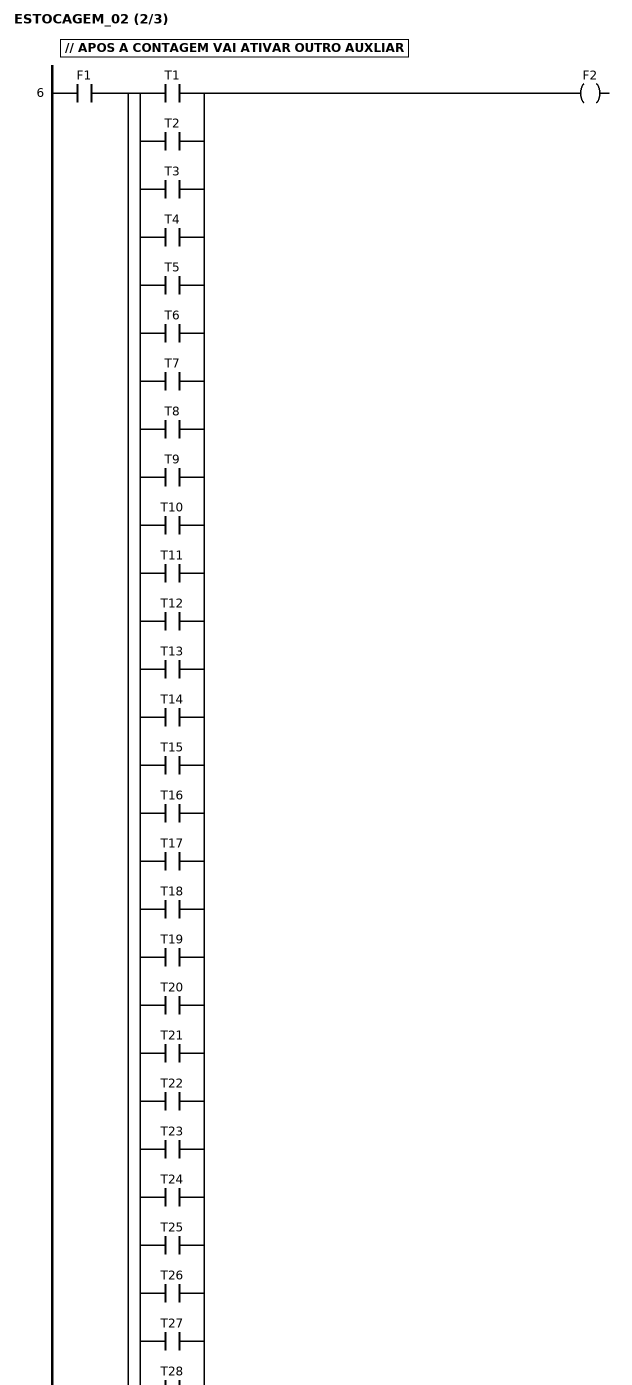
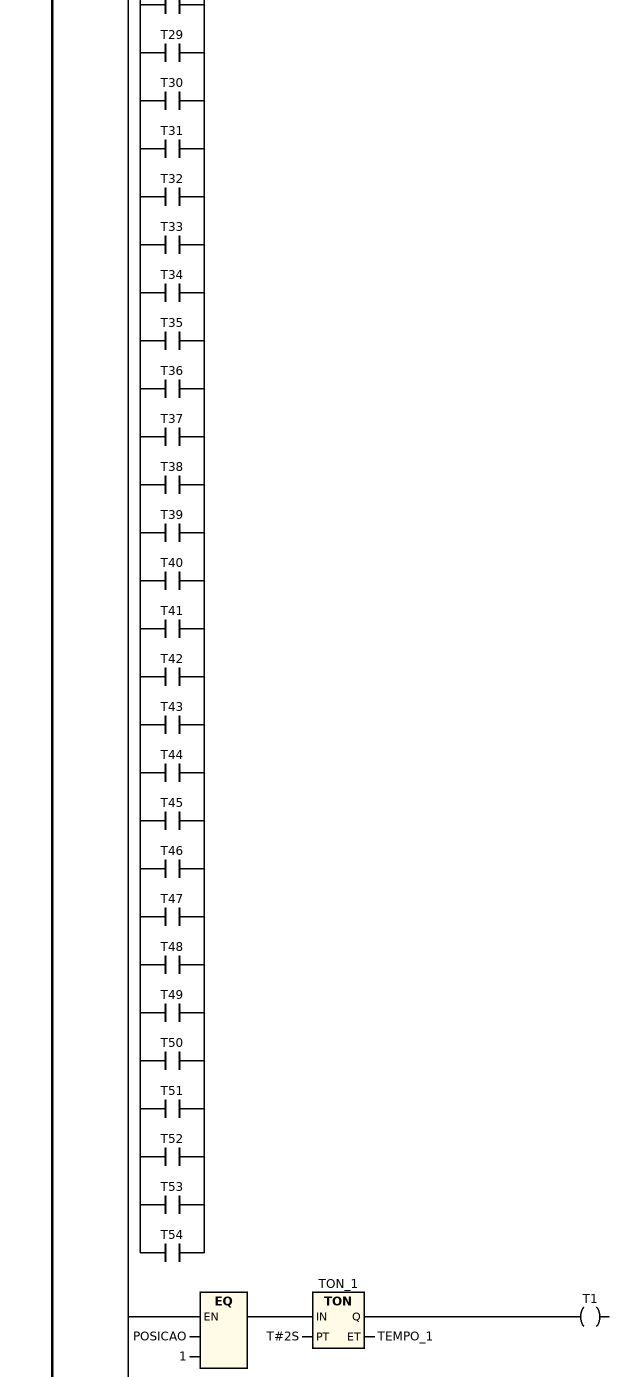
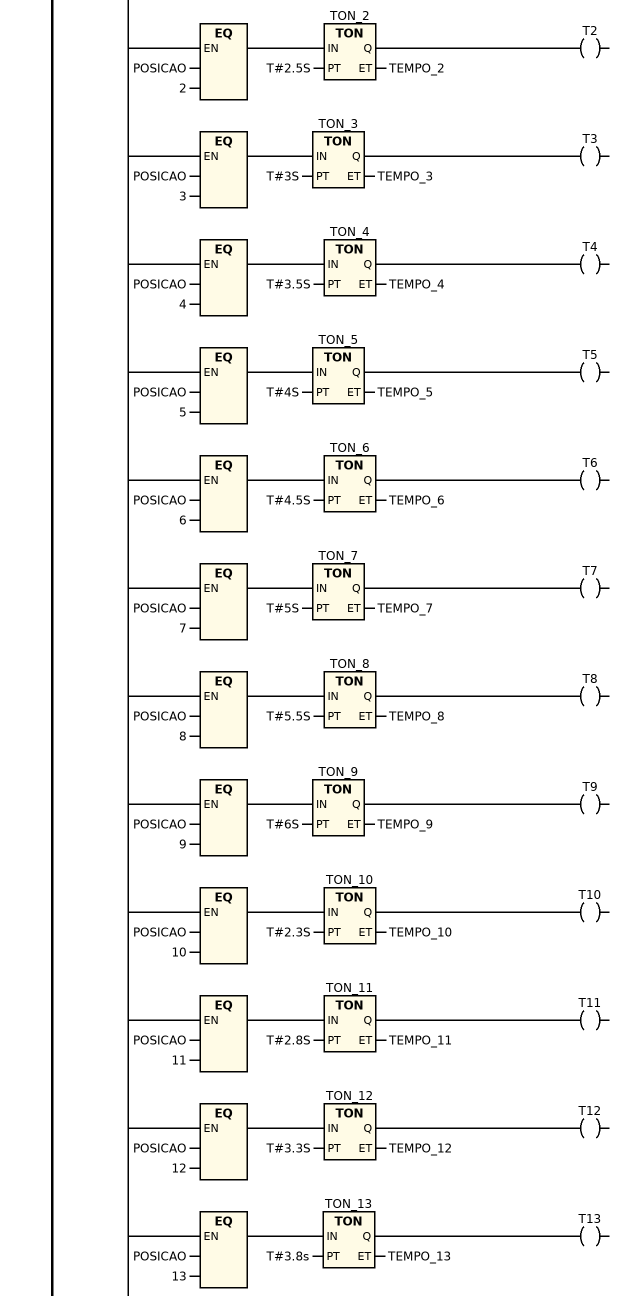
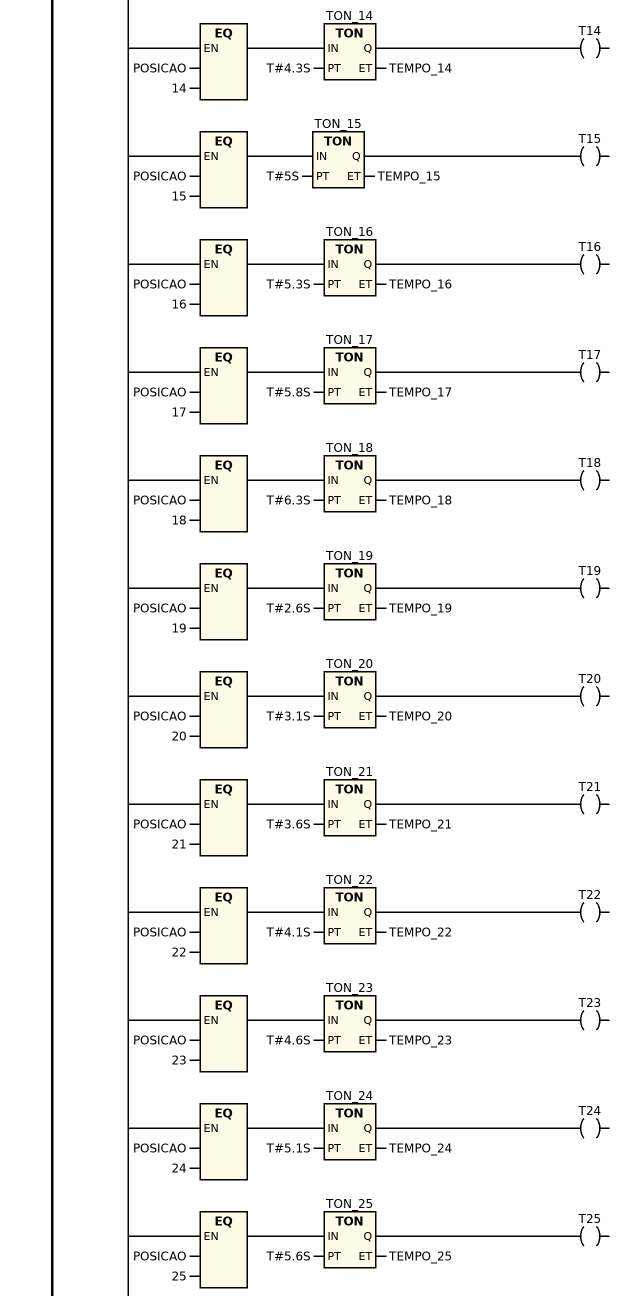
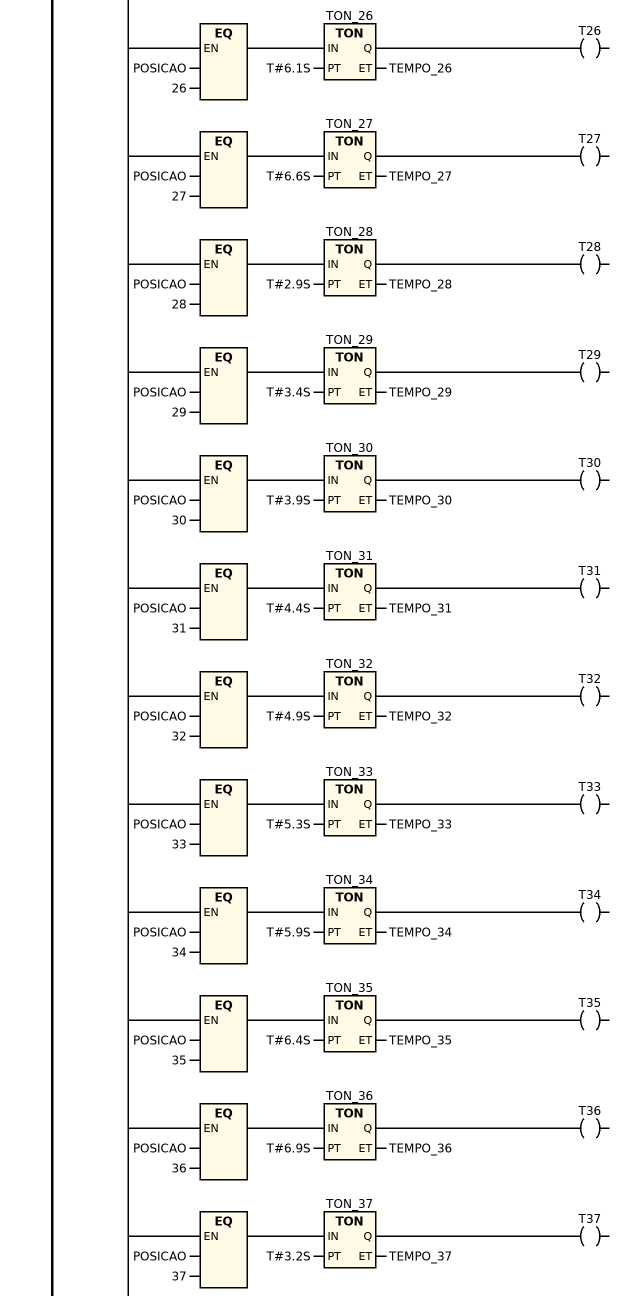
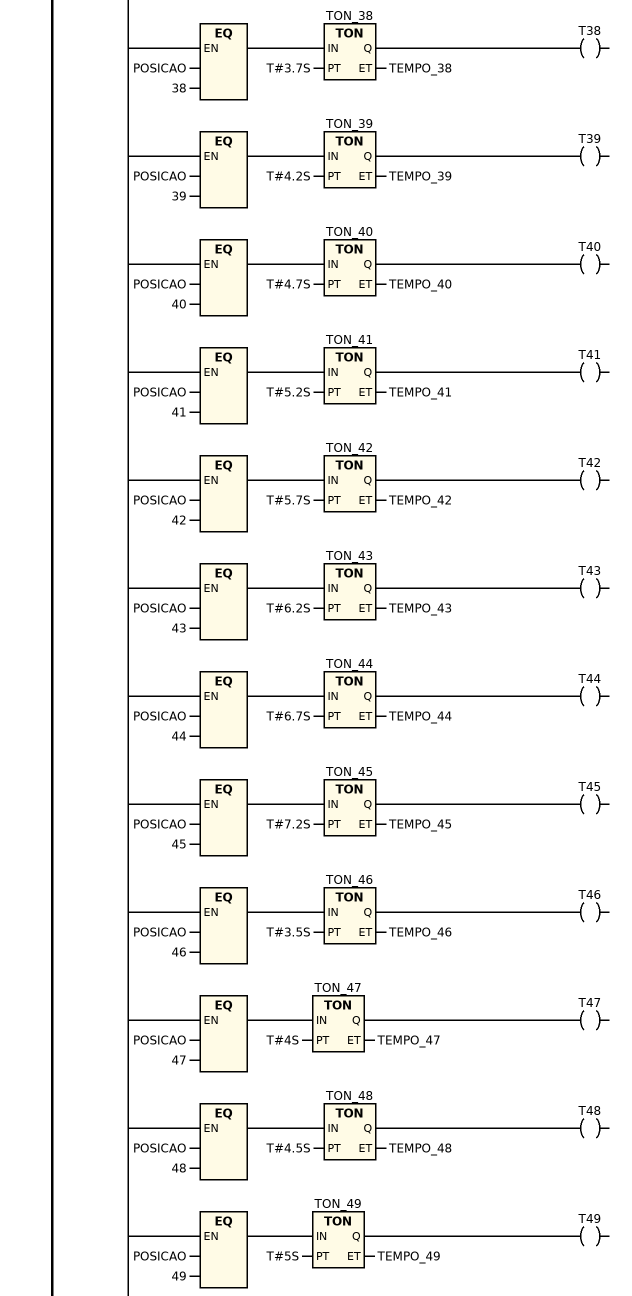
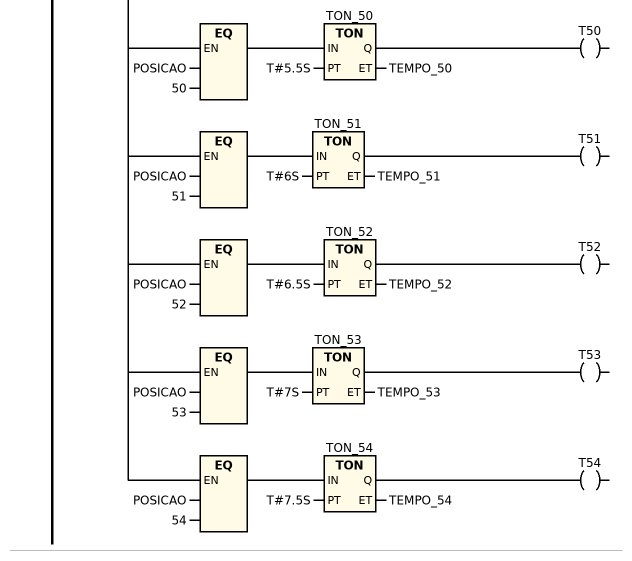
// NETWORK 6
// label: // APOS A CONTAGEM VAI ATIVAR OUTRO AUXLIAR
F2 := F1 AND (T1 OR T2 OR T3 OR T4 OR T5 OR T6 OR T7 OR T8 OR T9 OR T10 OR T11 OR T12 OR T13 OR T14 OR T15 OR T16 OR T17 OR T18 OR T19 OR T20 OR T21 OR T22 OR T23 OR T24 OR T25 OR T26 OR T27 OR T28 OR T29 OR T30 OR T31 OR T32 OR T33 OR T34 OR T35 OR T36 OR T37 OR T38 OR T39 OR T40 OR T41 OR T42 OR T43 OR T44 OR T45 OR T46 OR T47 OR T48 OR T49 OR T50 OR T51 OR T52 OR T53 OR T54);
TON_1(IN := F1 AND POSICAO = 1, PT := T#2S, ET => TEMPO_1); // TON
T1 := TON_1.Q;
TON_2(IN := F1 AND POSICAO = 2, PT := T#2.5S, ET => TEMPO_2); // TON
T2 := TON_2.Q;
TON_3(IN := F1 AND POSICAO = 3, PT := T#3S, ET => TEMPO_3); // TON
T3 := TON_3.Q;
TON_4(IN := F1 AND POSICAO = 4, PT := T#3.5S, ET => TEMPO_4); // TON
T4 := TON_4.Q;
TON_5(IN := F1 AND POSICAO = 5, PT := T#4S, ET => TEMPO_5); // TON
T5 := TON_5.Q;
TON_6(IN := F1 AND POSICAO = 6, PT := T#4.5S, ET => TEMPO_6); // TON
T6 := TON_6.Q;
TON_7(IN := F1 AND POSICAO = 7, PT := T#5S, ET => TEMPO_7); // TON
T7 := TON_7.Q;
TON_8(IN := F1 AND POSICAO = 8, PT := T#5.5S, ET => TEMPO_8); // TON
T8 := TON_8.Q;
TON_9(IN := F1 AND POSICAO = 9, PT := T#6S, ET => TEMPO_9); // TON
T9 := TON_9.Q;
TON_10(IN := F1 AND POSICAO = 10, PT := T#2.3S, ET => TEMPO_10); // TON
T10 := TON_10.Q;
TON_11(IN := F1 AND POSICAO = 11, PT := T#2.8S, ET => TEMPO_11); // TON
T11 := TON_11.Q;
TON_12(IN := F1 AND POSICAO = 12, PT := T#3.3S, ET => TEMPO_12); // TON
T12 := TON_12.Q;
TON_13(IN := F1 AND POSICAO = 13, PT := T#3.8s, ET => TEMPO_13); // TON
T13 := TON_13.Q;
TON_14(IN := F1 AND POSICAO = 14, PT := T#4.3S, ET => TEMPO_14); // TON
T14 := TON_14.Q;
TON_15(IN := F1 AND POSICAO = 15, PT := T#5S, ET => TEMPO_15); // TON
T15 := TON_15.Q;
TON_16(IN := F1 AND POSICAO = 16, PT := T#5.3S, ET => TEMPO_16); // TON
T16 := TON_16.Q;
TON_17(IN := F1 AND POSICAO = 17, PT := T#5.8S, ET => TEMPO_17); // TON
T17 := TON_17.Q;
TON_18(IN := F1 AND POSICAO = 18, PT := T#6.3S, ET => TEMPO_18); // TON
T18 := TON_18.Q;
TON_19(IN := F1 AND POSICAO = 19, PT := T#2.6S, ET => TEMPO_19); // TON
T19 := TON_19.Q;
TON_20(IN := F1 AND POSICAO = 20, PT := T#3.1S, ET => TEMPO_20); // TON
T20 := TON_20.Q;
TON_21(IN := F1 AND POSICAO = 21, PT := T#3.6S, ET => TEMPO_21); // TON
T21 := TON_21.Q;
TON_22(IN := F1 AND POSICAO = 22, PT := T#4.1S, ET => TEMPO_22); // TON
T22 := TON_22.Q;
TON_23(IN := F1 AND POSICAO = 23, PT := T#4.6S, ET => TEMPO_23); // TON
T23 := TON_23.Q;
TON_24(IN := F1 AND POSICAO = 24, PT := T#5.1S, ET => TEMPO_24); // TON
T24 := TON_24.Q;
TON_25(IN := F1 AND POSICAO = 25, PT := T#5.6S, ET => TEMPO_25); // TON
T25 := TON_25.Q;
TON_26(IN := F1 AND POSICAO = 26, PT := T#6.1S, ET => TEMPO_26); // TON
T26 := TON_26.Q;
TON_27(IN := F1 AND POSICAO = 27, PT := T#6.6S, ET => TEMPO_27); // TON
T27 := TON_27.Q;
TON_28(IN := F1 AND POSICAO = 28, PT := T#2.9S, ET => TEMPO_28); // TON
T28 := TON_28.Q;
TON_29(IN := F1 AND POSICAO = 29, PT := T#3.4S, ET => TEMPO_29); // TON
T29 := TON_29.Q;
TON_30(IN := F1 AND POSICAO = 30, PT := T#3.9S, ET => TEMPO_30); // TON
T30 := TON_30.Q;
TON_31(IN := F1 AND POSICAO = 31, PT := T#4.4S, ET => TEMPO_31); // TON
T31 := TON_31.Q;
TON_32(IN := F1 AND POSICAO = 32, PT := T#4.9S, ET => TEMPO_32); // TON
T32 := TON_32.Q;
TON_33(IN := F1 AND POSICAO = 33, PT := T#5.3S, ET => TEMPO_33); // TON
T33 := TON_33.Q;
TON_34(IN := F1 AND POSICAO = 34, PT := T#5.9S, ET => TEMPO_34); // TON
T34 := TON_34.Q;
TON_35(IN := F1 AND POSICAO = 35, PT := T#6.4S, ET => TEMPO_35); // TON
T35 := TON_35.Q;
TON_36(IN := F1 AND POSICAO = 36, PT := T#6.9S, ET => TEMPO_36); // TON
T36 := TON_36.Q;
TON_37(IN := F1 AND POSICAO = 37, PT := T#3.2S, ET => TEMPO_37); // TON
T37 := TON_37.Q;
TON_38(IN := F1 AND POSICAO = 38, PT := T#3.7S, ET => TEMPO_38); // TON
T38 := TON_38.Q;
TON_39(IN := F1 AND POSICAO = 39, PT := T#4.2S, ET => TEMPO_39); // TON
T39 := TON_39.Q;
TON_40(IN := F1 AND POSICAO = 40, PT := T#4.7S, ET => TEMPO_40); // TON
T40 := TON_40.Q;
TON_41(IN := F1 AND POSICAO = 41, PT := T#5.2S, ET => TEMPO_41); // TON
T41 := TON_41.Q;
TON_42(IN := F1 AND POSICAO = 42, PT := T#5.7S, ET => TEMPO_42); // TON
T42 := TON_42.Q;
TON_43(IN := F1 AND POSICAO = 43, PT := T#6.2S, ET => TEMPO_43); // TON
T43 := TON_43.Q;
TON_44(IN := F1 AND POSICAO = 44, PT := T#6.7S, ET => TEMPO_44); // TON
T44 := TON_44.Q;
TON_45(IN := F1 AND POSICAO = 45, PT := T#7.2S, ET => TEMPO_45); // TON
T45 := TON_45.Q;
TON_46(IN := F1 AND POSICAO = 46, PT := T#3.5S, ET => TEMPO_46); // TON
T46 := TON_46.Q;
TON_47(IN := F1 AND POSICAO = 47, PT := T#4S, ET => TEMPO_47); // TON
T47 := TON_47.Q;
TON_48(IN := F1 AND POSICAO = 48, PT := T#4.5S, ET => TEMPO_48); // TON
T48 := TON_48.Q;
TON_49(IN := F1 AND POSICAO = 49, PT := T#5S, ET => TEMPO_49); // TON
T49 := TON_49.Q;
TON_50(IN := F1 AND POSICAO = 50, PT := T#5.5S, ET => TEMPO_50); // TON
T50 := TON_50.Q;
TON_51(IN := F1 AND POSICAO = 51, PT := T#6S, ET => TEMPO_51); // TON
T51 := TON_51.Q;
TON_52(IN := F1 AND POSICAO = 52, PT := T#6.5S, ET => TEMPO_52); // TON
T52 := TON_52.Q;
TON_53(IN := F1 AND POSICAO = 53, PT := T#7S, ET => TEMPO_53); // TON
T53 := TON_53.Q;
TON_54(IN := F1 AND POSICAO = 54, PT := T#7.5S, ET => TEMPO_54); // TON
T54 := TON_54.Q;

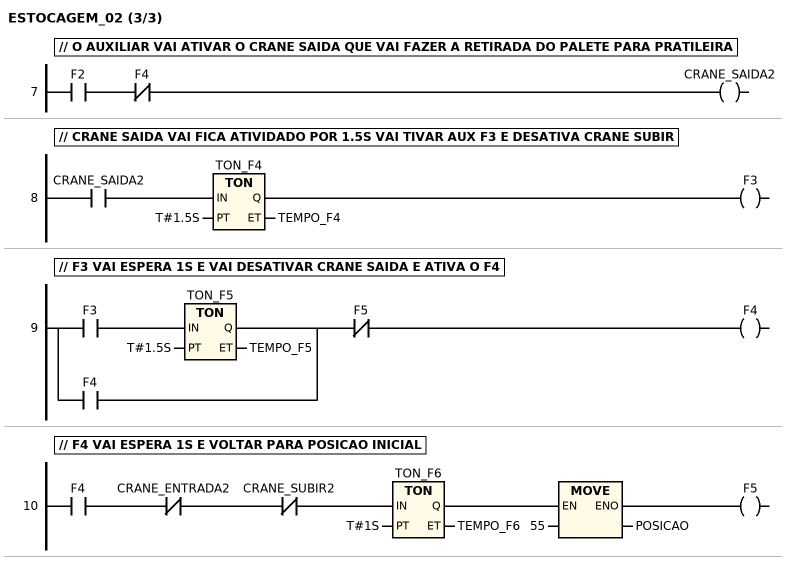
// NETWORK 7
// label: // O AUXILIAR VAI ATIVAR O CRANE SAIDA QUE VAI FAZER A RETIRADA DO PALETE PARA PRATILEIRA
CRANE_SAIDA2 := F2 AND NOT F4;

// NETWORK 8
// label: // CRANE SAIDA VAI FICA ATIVIDADO POR 1.5S VAI TIVAR AUX F3 E DESATIVA CRANE SUBIR
TON_F4(IN := CRANE_SAIDA2, PT := T#1.5S, ET => TEMPO_F4); // TON
F3 := TON_F4.Q;

// NETWORK 9
// label: // F3 VAI ESPERA 1S E VAI DESATIVAR CRANE SAIDA E ATIVA O F4
TON_F5(IN := F3, PT := T#1.5S, ET => TEMPO_F5); // TON
F4 := (TON_F5.Q OR F4) AND NOT F5;

// NETWORK 10
// label: // F4 VAI ESPERA 1S E VOLTAR PARA POSICAO INICIAL
TON_F6(IN := F4 AND NOT CRANE_ENTRADA2 AND NOT CRANE_SUBIR2, PT := T#1S, ET => TEMPO_F6); // TON
_w3 := TON_F6.Q;
IF _w3 THEN POSICAO := 55; END_IF
F5 := _w3;

END_PROGRAM

// Device/Application/VACUO_02
PROGRAM VACUO_02
VAR	
// ESTEIRA SECUDARIA N 02(AZUL)
	//ENTRADAS
	_SENSOR_SAIDA02:BOOL;
	
	//SAIDAS
	ESTEIRA_SECUDARIA02:BOOL;
	ESTEIRA_CURVA_SECUNDARIA2: BOOL;
	ESTEIRA_CURVA_SECUNDARIA2_1: BOOL;
	ESTEIRA_SAIDA_PALETE2: BOOL;
	CONTAGEM_AZUIS: UINT;
	
// VACUO N 02
	//ENTRADAS
	_SENSOR_ENTRADA02:BOOL;
	_DETECTED_VACUO02:BOOL;
	
	//SAIDAS
	X2:BOOL;
	Y2:BOOL;
	VACUO_2:BOOL;
	
// AUXILIARES
	CAIXA_AZUL: BOOL;
	B1: BOOL;
	B2: BOOL;
	B3: BOOL;
	B4: BOOL;
	B5: BOOL;
	B6: BOOL;
	B7: BOOL;
	B8: BOOL;
	B9: BOOL;
	B10: BOOL;
	B11: BOOL;
	B12:BOOL;
	
//TEMPORIZADORES
	TON_1B: TON;
	TEMPO_1B: TIME;
	TON_2B: TON;
	TEMPO_2B: TIME;
	TON_3B: TON;
	TEMPO_3B: TIME;
	TON_4B: TON;
	TEMPO_4B: TIME;
	TON_5B: TON;
	TEMPO_5B: TIME;
	TON_6B: TON;
	TEMPO_6B: TIME;
	TON_7B: TON;
	TEMPO_7B: TIME;
	TON_8B: TON;
	TEMPO_8B: TIME;
	TON_9B: TON;
	TEMPO_9B: TIME;
	TON_10B: TON;
	TEMPO_10B: TIME;
	CTU_1B: CTU;
	CONT_1B: WORD;
END_VAR
VAR // added by the converter: edge detectors and wires of the graphical bodies
    _w1, _w2, _w3, _w4 : BOOL;
END_VAR

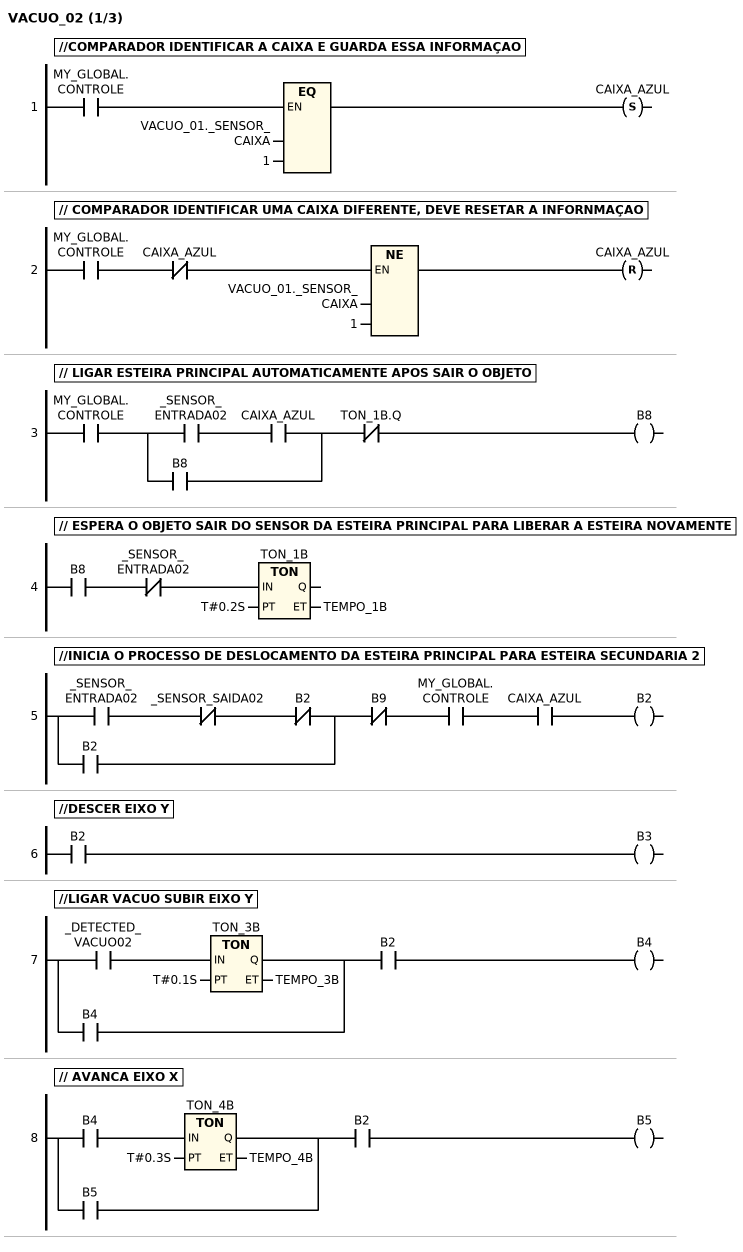
// NETWORK 1
// label: //COMPARADOR IDENTIFICAR A CAIXA E GUARDA ESSA INFORMAÇAO
CAIXA_AZUL S= MY_GLOBAL.CONTROLE AND VACUO_01._SENSOR_CAIXA = 1;

// NETWORK 2
// label: // COMPARADOR IDENTIFICAR UMA CAIXA DIFERENTE, DEVE RESETAR A INFORNMAÇAO
CAIXA_AZUL R= MY_GLOBAL.CONTROLE AND NOT CAIXA_AZUL AND VACUO_01._SENSOR_CAIXA <> 1;

// NETWORK 3
// label: // LIGAR ESTEIRA PRINCIPAL AUTOMATICAMENTE APOS SAIR O OBJETO
B8 := MY_GLOBAL.CONTROLE AND (_SENSOR_ENTRADA02 AND CAIXA_AZUL OR B8) AND NOT TON_1B.Q;

// NETWORK 4
// label: // ESPERA O OBJETO SAIR DO SENSOR DA ESTEIRA PRINCIPAL PARA LIBERAR A ESTEIRA NOVAMENTE
TON_1B(IN := B8 AND NOT _SENSOR_ENTRADA02, PT := T#0.2S, ET => TEMPO_1B); // TON

// NETWORK 5
// label: //INICIA O PROCESSO DE DESLOCAMENTO DA ESTEIRA PRINCIPAL PARA ESTEIRA SECUNDARIA 2
B2 := (_SENSOR_ENTRADA02 AND NOT _SENSOR_SAIDA02 AND NOT B2 OR B2) AND NOT B9 AND MY_GLOBAL.CONTROLE AND CAIXA_AZUL;

// NETWORK 6
// label: //DESCER EIXO Y
B3 := B2;

// NETWORK 7
// label: //LIGAR VACUO SUBIR EIXO Y
TON_3B(IN := _DETECTED_VACUO02, PT := T#0.1S, ET => TEMPO_3B); // TON
B4 := (TON_3B.Q OR B4) AND B2;

// NETWORK 8
// label: // AVANCA EIXO X
TON_4B(IN := B4, PT := T#0.3S, ET => TEMPO_4B); // TON
B5 := (TON_4B.Q OR B5) AND B2;

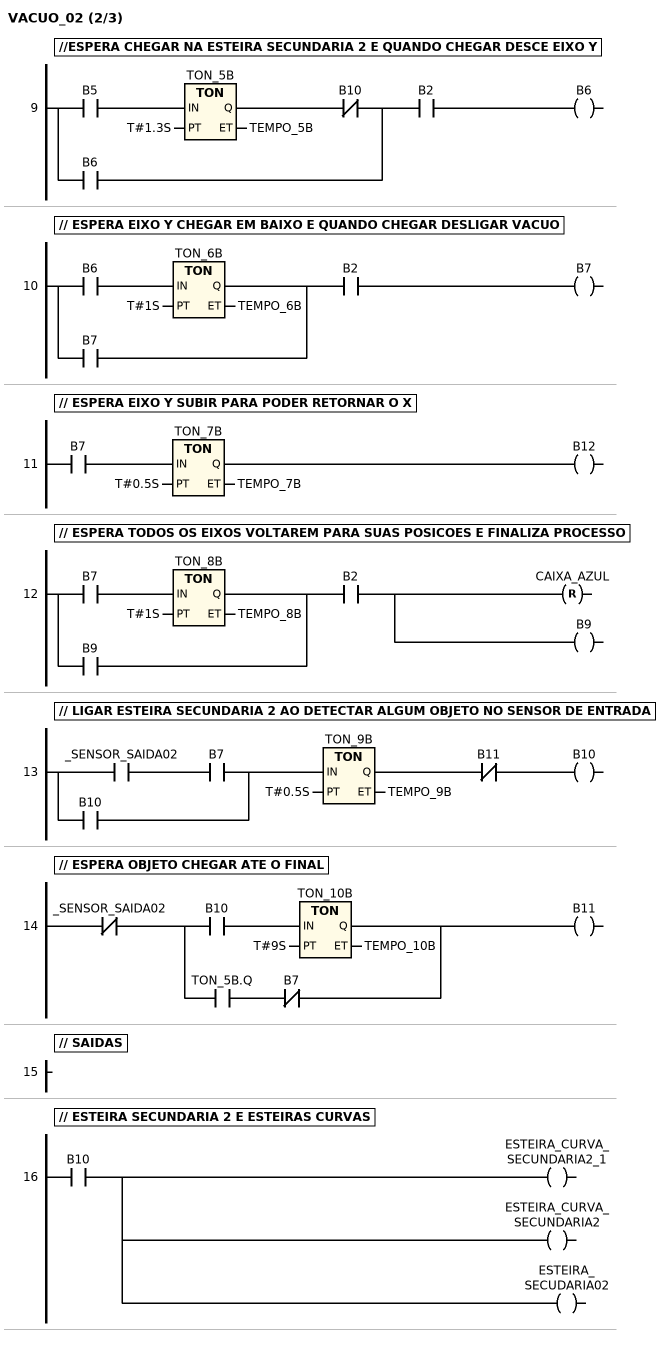
// NETWORK 9
// label: //ESPERA CHEGAR NA ESTEIRA SECUNDARIA 2 E QUANDO CHEGAR DESCE EIXO Y
TON_5B(IN := B5, PT := T#1.3S, ET => TEMPO_5B); // TON
B6 := (TON_5B.Q AND NOT B10 OR B6) AND B2;

// NETWORK 10
// label: // ESPERA EIXO Y CHEGAR EM BAIXO E QUANDO CHEGAR DESLIGAR VACUO
TON_6B(IN := B6, PT := T#1S, ET => TEMPO_6B); // TON
B7 := (TON_6B.Q OR B7) AND B2;

// NETWORK 11
// label: // ESPERA EIXO Y SUBIR PARA PODER RETORNAR O X
TON_7B(IN := B7, PT := T#0.5S, ET => TEMPO_7B); // TON
B12 := TON_7B.Q;

// NETWORK 12
// label: // ESPERA TODOS OS EIXOS VOLTAREM PARA SUAS POSICOES E FINALIZA PROCESSO
TON_8B(IN := B7, PT := T#1S, ET => TEMPO_8B); // TON
_w1 := (TON_8B.Q OR B9) AND B2;
CAIXA_AZUL R= _w1;
B9 := _w1;

// NETWORK 13
// label: // LIGAR ESTEIRA SECUNDARIA 2 AO DETECTAR ALGUM OBJETO NO SENSOR DE ENTRADA
TON_9B(IN := _SENSOR_SAIDA02 AND B7 OR B10, PT := T#0.5S, ET => TEMPO_9B); // TON
B10 := TON_9B.Q AND NOT B11;

// NETWORK 14
// label: // ESPERA OBJETO CHEGAR ATE O FINAL
_w2 := NOT _SENSOR_SAIDA02;
_w3 := (_w2 AND TON_5B.Q) AND NOT B7;
IF NOT _w3 THEN
    TON_10B(IN := _w2 AND B10, PT := T#9S, ET => TEMPO_10B); // TON
    _w3 := TON_10B.Q;
END_IF
B11 := _w3;

// NETWORK 15
// label: // SAIDAS

// NETWORK 16
// label: // ESTEIRA SECUNDARIA 2 E ESTEIRAS CURVAS
ESTEIRA_CURVA_SECUNDARIA2_1 := B10;
ESTEIRA_CURVA_SECUNDARIA2 := B10;
ESTEIRA_SECUDARIA02 := B10;

